IF xFalha THEN
	CASE wFalha OF
		16#0:
			sStatusConexao := 'Inversor Offline';
			xInversorOnline := FALSE;
		16#1080:
			sStatusConexao := 'Tempo Limite Backup/Restauração';
		16#1081:
			sStatusConexao := 'Falha na classificação do ID';
		16#2281:
			sStatusConexao := 'Calibração';
		16#2310:
			sStatusConexao := 'Sobrecorrente';
		16#2330:
			sStatusConexao := 'Fuga à Terra';
		16#2340:
			sStatusConexao := 'Curto-Circuito na Saída';
		16#2381:
			sStatusConexao := 'Sobrecarga no IGBT';
		16#3130:
			sStatusConexao := 'Falta de Fase na Entrada';
		16#3181:
			sStatusConexao := 'Cross Connection';
		16#3210:
			sStatusConexao := 'Sobretensão CC no Circuito intermediário';
		16#3220:
			sStatusConexao := 'Subtensão CC no Circuito intermediário';
		16#3381:
			sStatusConexao := 'Falta de Fase na Saída';
		16#4110:
			sStatusConexao := 'Temperatura alta na placa de controle';
		16#4210:
			sStatusConexao := 'Sobretemperatura estimada no IGBT';
		16#4290:
			sStatusConexao := 'Temperatura alta no módulo do inversor';
		16#42F1:
			sStatusConexao := 'Sobretemperatura no IGBT';
		16#4310:
			sStatusConexao := 'Temperatura alta no módulo de potência';
		16#4380:
			sStatusConexao := 'Diferença de temperatura IGBT';
		16#4981:
			sStatusConexao := 'Falha - Temperatura externa 1';
		16#4982:
			sStatusConexao := 'Falha - Temperatura externa 2';
		16#5090:
			sStatusConexao := 'Falha no Hardware STO';
		16#5091:
			sStatusConexao := 'STO - Safe Torque OFF';
		16#5092:
			sStatusConexao := 'Erro Lógico PU';
		16#5093:
			sStatusConexao := 'Hardware incompatível com Firmware';
		16#5094:
			sStatusConexao := 'Falha na Medição de Temperatura interna';
		16#50A0:
			sStatusConexao := 'Ventilador de Refrigeração em Falha';
		16#5681:
			sStatusConexao := 'Falha na comunicação PU';
		16#5682:
			sStatusConexao := 'Unidade de Potência Perdida';
		16#5690:
			sStatusConexao := 'Falha na Comunicação Interna';
		16#5691:
			sStatusConexao := 'Falha no Circuito de Medição';
		16#5692:
			sStatusConexao := 'Falha de Alimentação na Unidade de Potência';
		16#5693:
			sStatusConexao := 'Falha no Circuito de Medição';
		16#5696:
			sStatusConexao := 'Feedback dos Estados das Fases Incorreto';
		16#5697:
			sStatusConexao := 'Sem sinal de Feedback das Fases';
		16#6181:
			sStatusConexao := 'Versão da FPGA incompatível com o Firmware';
		16#6306:
			sStatusConexao := 'Sem sinal de Feedback das Fases';
		16#6481:
			sStatusConexao := 'Falha Interna';
		16#6487:
			sStatusConexao := 'Falha Interna';
		16#64A1:
			sStatusConexao := 'Erro de Leitura de Arquivo';
		16#64A6:
			sStatusConexao := 'Falha no programa adaptativo';
		16#64B2:
			sStatusConexao := 'Falha no conjunto de parâmetros utilizados';
		16#64E1:
			sStatusConexao := 'Erro de Sistema Operacional';
		16#6581:
			sStatusConexao := 'Falha ao salvar/carregar parâmetro';
		16#65A1:
			sStatusConexao := 'Informação requerida pelo PLC não disponpivel';
		16#6681:
			sStatusConexao := 'Perda comunicação EFB(FieldBus Integrado)';
		16#6682:
			sStatusConexao := 'Falha ao ler o arquivo EFB(FieldBus Integrado)';
		16#6683:
			sStatusConexao := 'Parâmetro EFB(FieldBus Integrado) inválido';
		16#6684:
			sStatusConexao := 'Falha ao carregar o firmware EFB(FieldBus Integrado)';
		16#6685:
			sStatusConexao := 'Falha reservada EFB(FieldBus Integrado) 1';
		16#6686:
			sStatusConexao := 'Falha reservada EFB(FieldBus Integrado) 2';
		16#6882:
			sStatusConexao := 'Falha Interna';
		16#6885:
			sStatusConexao := 'Falha Interna';
		16#7081:
			sStatusConexao := 'Perda do Painel de Controle';
		16#7082:
			sStatusConexao := 'Perda de Comunicação do Módulo I/O';
		16#7086:
			sStatusConexao := 'Sobretensão no Módulo I/O';
		16#71A2:
			sStatusConexao := 'Falha de Controle do Freio Meânico (Fechamento)';
		16#71A3:
			sStatusConexao := 'Falha de Controle do Freio Meânico (Abertura)';
		16#71A5:
			sStatusConexao := 'Freio Mecânico Travado';
		16#7121:
			sStatusConexao := 'Motor bloqueado: Carga Excessiva ou Energia Insuficiente';
		16#7181:
			sStatusConexao := 'Problema na Resistência de Frenagem';
		16#7183:
			sStatusConexao := 'Temperatura Alta na Resistência de Frenagem';
		16#7184:
			sStatusConexao := 'Curto-Circuito na Resistência de Frenagem';
		16#7191:
			sStatusConexao := 'Curto-Circuito no Chopper IGBT';
		16#7192:
			sStatusConexao := 'Temperatura Alta no Chopper IGBT';
		16#7301:
			sStatusConexao := 'Sem Feedback de Velocidade do Motor';
		16#7310:
			sStatusConexao := 'Sobrevelocidade';
		16#7381:
			sStatusConexao := 'Falha no Feedback do Encoder';
		16#73F0:
			sStatusConexao := 'Sobrefrequência';
		16#73B0:
			sStatusConexao := 'Falha na Parada de Emergência';
		16#7510:
			sStatusConexao := 'Perda de comunicação FBA A';
		16#8001:
			sStatusConexao := 'Falha de subcarga (Abaixo)';
		16#8002:
			sStatusConexao := 'Falha de subcarga (Acima)';
		16#80A0:
			sStatusConexao := 'Sinal Analógico Fora dos Limites';
		16#80B0:
			sStatusConexao := 'Falha Supervisão de Sinal 66';
		16#80B1:
			sStatusConexao := 'Falha Supervisão de Sinal 66';
		16#80B2:
			sStatusConexao := 'Falha Supervisão de Sinal 66';
		16#80B3:
			sStatusConexao := 'Falha Supervisão de Sinal 66';
		16#80B4:
			sStatusConexao := 'Falha Supervisão de Sinal 66';
		16#80B5:
			sStatusConexao := 'Falha Supervisão de Sinal 66';
		16#9081:
			sStatusConexao := 'Falha Dispotivo Externo 1';
		16#9082:
			sStatusConexao := 'Falha Dispotivo Externo 2';
		16#9083:
			sStatusConexao := 'Falha Dispotivo Externo 3';
		16#9084:
			sStatusConexao := 'Falha Dispotivo Externo 4';
		16#9085:
			sStatusConexao := 'Falha Dispotivo Externo 5';
		16#FA81:
			sStatusConexao := 'STO (Safe Torque OFF) 1 rompido';
		16#FA82:
			sStatusConexao := 'STO (Safe Torque OFF) 1 rompido';
		16#FF61:
			sStatusConexao := 'ID Run';
		16#FF81:
			sStatusConexao := 'Falha forçada FBA';
		16#FF8E:
			sStatusConexao := 'Falha forçada FBB';
		16#D100:
			sStatusConexao := 'Inversor não Consegiu Fornecer Torque Suficiente';
		16#D101:
			sStatusConexao := 'Escorregamento do Freio';
		16#D102:
			sStatusConexao := 'Velocidade abaixo do limite de segurança';
		16#D105:
			sStatusConexao := 'Velocidade do motor Excedeu o Desvio De Estado Estacionário';
		16#D108:
			sStatusConexao := 'Comando de limite de parada Frente e Ré Ativos Simultaneamente';
	END_CASE
ELSE
	IF NOT xRun AND NOT Motor.Sa.xFalha THEN
		sStatusConexao := 'Pronto para Rodar';
	ELSE
		sStatusConexao := 'Rodando';
	END_IF
	
	IF Motor.Sa.xFalha THEN
		sStatusConexao := 'Inversor OK / Falha na Partida';
	END_IF
END_IF

IF xGuardaRegistroErro THEN
	xInversorOnline := FALSE;
END_IF
END_ACTION

END_FUNCTION_BLOCK

// POUs/Comunicação/ModbusRTU/FB_ModBusRTU_ALTISTAR22
{attribute 'hide_all_locals'}
FUNCTION_BLOCK FB_ModBusRTU_ALTISTAR22
VAR_IN_OUT
	MestreModbusRTU	: ModbusRtuMasterV2_KL6x22B;
	Motor			: st_Partida;
END_VAR
VAR_INPUT
	xInicia				: BOOL;
END_VAR
VAR_OUTPUT
	//Gerais
	xTerminei				: BOOL;
	UltimoModbusErro		: ST_ModbusErrorDiagnostics;
END_VAR
VAR
	xIniciaInterno				: BOOL;	
	xTerminouLeitura			: BOOL;
	xTerminouEscrita			: BOOL;
	xSoftOnline					: BOOL;
	xGuardaRegistroErro			: BOOL;
	ControlWord					:  WORD;

	
	iRegistradorAtual			: INT := 1;
	
	wLeitura					: WORD;
	rVelocidadeAux				: WORD;
	wFalha						: WORD;
	StatusWord					: WORD;
	arLeitura					: ARRAY[1..7] OF WORD;
	arEscrita					: ARRAY[1..3] OF WORD;
	
	RegistradoresLeitura		: ARRAY[1..7] OF INT 	:= [19,20,256,257,258,259,279];		//Registradores de leitura
	RegistradoresEscrita		: ARRAY[1..3] OF INT 	:= [19,20,752];		//Registradores de escrita
	
	stateModbus					: State_Modbus;			//Variável para máquina de estados
	state						: StateWord;
	
	rt							: R_TRIG;				//Inicia vindo de fora
	ft							: F_TRIG;				//Inicio vindo de fora
	rtInicia 					: R_TRIG;				//Inicia Leitura/Escrita
	ftInicia					: F_TRIG;				//Para Leitura/Escrita
	
	tTimeout					: TIME := T#1S;			//Tempo de timeout para espera escravo 
	tonTimeout					: TON;

	xFalha					: BOOL;
	xPronto					: BOOL;
	xRodando				: BOOL;
	sStatusConexao			: STRING;
	rCorrenteL1				: REAL;
	rCorrenteL2				: REAL;
	rCorrenteL3				: REAL;
	rTempoACCAtual			: REAL;
	rTempoDECAtual			: REAL;
	
	iEndereco 			: INT;
END_VAR

IF xLicensaValida5154156 THEN
	rt(CLK := xInicia, Q =>);
	
	IF rt.Q THEN
		xIniciaInterno := TRUE;
	END_IF
	
	
	rtInicia(CLK := xIniciaInterno, Q =>);
	ftInicia(CLK := xIniciaInterno, Q =>);
	
	IF rtInicia.Q THEN
		iRegistradorAtual	:= 1;
		xTerminei			:= FALSE;
		
		//Quando inicia a leitura, não terminou de ler nenhum
		xTerminouLeitura	:= FALSE;
		xTerminouEscrita	:= FALSE;
		
		stateModbus := State_Modbus.Inicia;
	END_IF
	
	IF ftInicia.Q  THEN
		xIniciaInterno := FALSE;
		xInicia := FALSE;
		iRegistradorAtual := 1;
		xTerminei := TRUE;
		MestreModbusRTU.ReadRegs(Execute := FALSE);
		MestreModbusRTU.WriteRegs(Execute := FALSE);
	END_IF
	
	EspelhoEntradas();
	
	Leitura();
	
	Estados();
	
	ExecutaEstados();
	
	Status();
	
	EspelhoSaidas();
	
	Escrita();
	
	tonTimeOut(IN:= MestreModbusRTU.BUSY, PT:= T#10S, Q=> , ET=> );
	
	IF tonTimeOut.Q THEN
		//xIniciaInterno := FALSE;
		//xInicia := FALSE;
	END_IF

ELSE
	ValidaLicensa();
END_IF

ACTION Escrita:
CASE stateModbus OF
	
	State_Modbus.Inicia:
		IF xIniciaInterno THEN
			MestreModbusRTU.ReadRegs(Execute := FALSE);
			MestreModbusRTU.WriteSingleCoil(Execute := FALSE);

			//Se não terminou de ler corrente, fica lendo a corrente	
			IF NOT xTerminouLeitura THEN
				stateModbus := State_Modbus.Leitura;
			ELSE
				IF NOT xTerminouEscrita THEN
					stateModbus := State_Modbus.Escrita;
				END_IF
			END_IF;

			IF xTerminouLeitura AND xTerminouEscrita THEN
				xIniciaInterno := FALSE;
				xTerminei := TRUE;
			END_IF
		END_IF
			
	State_Modbus.Escrita:
	
		MestreModbusRTU.WriteSingleRegister(
			UnitID      := TO_BYTE(iEndereco),                 					// Endereço do equipamento escravo na rede Modbus
			Quantity    := 1,                									// Quantidade de WORDs a serem lidas
			MBAddr      := TO_WORD(RegistradoresEscrita[iRegistradorAtual]),	// Endereço Modbus. Onde 0 = Holding Register 40001
			cbLength    := SIZEOF(arEscrita[iRegistradorAtual]), 				// Quantidade de bytes a serem lidos
			pMemoryAddr := ADR(arEscrita[iRegistradorAtual]),					// Ponteiro para o array que receberá os dados lidos
			Execute     := TRUE,              									// Comando para executar o comando    
			Timeout     := tTimeout               								// Tempo de espera da resposta do escravo
		);

		IF NOT MestreModbusRTU.BUSY THEN
			IF MestreModbusRTU.Error THEN
				//Se deu erro cai fora
						xTerminouLeitura	:= TRUE;
						xTerminouEscrita	:= TRUE;
						
						stateModbus := State_Modbus.Inicia;
						xIniciaInterno := FALSE;
						
						xGuardaRegistroErro := TRUE;
			END_IF
			
			MestreModbusRTU.WriteSingleRegister(Execute := FALSE);
	
			stateModbus := State_Modbus.Inicia;		
			
			iRegistradorAtual := iRegistradorAtual + 1;	
			
			IF iRegistradorAtual > 3 THEN
				stateModbus := State_Modbus.Inicia;
				iRegistradorAtual := 1;
				xTerminouEscrita	:= TRUE;
				
				xGuardaRegistroErro := FALSE;
			END_IF

		END_IF 
END_CASE
END_ACTION

ACTION EspelhoEntradas:




arEscrita[1]	:= REAL_TO_WORD(Motor.Config.inversor.ACC);
arEscrita[2]	:= REAL_TO_WORD(Motor.Config.inversor.DEC);
arEscrita[3]	:= ControlWord;
iEndereco		:= Motor.En.i;

IF arEscrita[1] = 0 THEN
	arEscrita[1] := 1;
END_IF
END_ACTION

ACTION EspelhoSaidas:
StatusWord				:= arLeitura[3];
wFalha					:= arLeitura[7];

CASE wFalha OF
		1:
			Motor.Sa.sUltimoErro := 'Subcarga do Motor (Subcorrente) [UCF]';
		2:
			Motor.Sa.sUltimoErro := 'Sobrecorrente do Motor [OCF]';
		3:
			Motor.Sa.sUltimoErro := 'Desequilibrio de Fase [PHBD]';
		4:
			Motor.Sa.sUltimoErro := 'Detec. Corrente de Fuga à Terra Falha [GRDF]';
		5:
			Motor.Sa.sUltimoErro := 'Sobrecarga do Motor [OLF]';
		6:
			Motor.Sa.sUltimoErro := 'Temperatura Excessiva do Motor [OTF]';
		7:
			Motor.Sa.sUltimoErro := 'Falha Dectada de Sobreaquecimento [OHF]';
		8:
			Motor.Sa.sUltimoErro := 'Inversão de Fase [PIF]';
		9:
			Motor.Sa.sUltimoErro := 'Perda de Fase da Rede [PHF]';
		10:
			Motor.Sa.sUltimoErro := 'Subtensão ou Falta de Tensão [USF]';
		11:
			Motor.Sa.sUltimoErro := 'Sobretensão [OSF]';
		12:
			Motor.Sa.sUltimoErro := 'Falha Detectada de Tempo de Partida [STF]';
		13:
			Motor.Sa.sUltimoErro := 'Números de Partidas Excedido [SNBF]';
		14:
			Motor.Sa.sUltimoErro := 'Tiristor em Curto ou Conexão Incorreta [SSCR]';
		15:
			Motor.Sa.sUltimoErro := 'Falha Externa Detectada [ETF]';
		16:
			Motor.Sa.sUltimoErro := 'Falha Interna Detectada [INF]';
		17:
			Motor.Sa.sUltimoErro := 'Intervalo de Tempo Modbus [SLF]';
		18:
			Motor.Sa.sUltimoErro := 'Trap Code [TRAP]';
		19:
			Motor.Sa.sUltimoErro := 'Curto Circuito [SCF]';
		20:
			Motor.Sa.sUltimoErro := 'Falha Dectada Contador de By-Pass [BPF]';
		21:
			Motor.Sa.sUltimoErro := 'Config. Inválida na Energização [CFF]';
END_CASE

UltimoModbusErro			:= MestreModbusRTU.ErrorDiagnostics;
Motor.Sa.sStatusConexao		:= sStatusConexao;
Motor.En.xContatoFalhaSoft	:= xFalha AND NOT Motor.Config.xBypassRede;
Motor.Config.xTemSoft		:= TRUE;
Motor.En.xSoftOnline		:= xSoftOnline;

rTempoACCAtual			:= WORD_TO_REAL(arLeitura[1]);
rTempoDECAtual			:= WORD_TO_REAL(arLeitura[2]);
Motor.Sa.rCorrente		:= WORD_TO_REAL(arLeitura[4]);
rCorrenteL2				:= WORD_TO_REAL(arLeitura[5]);
rCorrenteL3				:= WORD_TO_REAL(arLeitura[6]);
END_ACTION

ACTION Estados:
//Rdy
IF StatusWord.0 THEN
	xPronto	:= TRUE;
ELSE
	xPronto	:= FALSE;
END_IF

//Run
IF StatusWord.1 THEN
	xRodando := TRUE;
ELSE
	xRodando := FALSE;
END_IF

//Falha
IF StatusWord.2 OR NOT StatusWord.0 THEN
	xFalha	:= TRUE;
ELSE
	xFalha	:= FALSE;
END_IF

StatusWord.0;
StatusWord.1;
StatusWord.2;
StatusWord.3;
StatusWord.4;
StatusWord.5;
StatusWord.6;
StatusWord.7;
StatusWord.8;
StatusWord.9;
StatusWord.10;
StatusWord.11;
StatusWord.12;
StatusWord.13;
StatusWord.14;
StatusWord.15;
END_ACTION

ACTION ExecutaEstados:
IF Motor.Sa.xCmdFwd THEN
	ControlWord := 1;
END_IF

IF NOT Motor.Sa.xCmdFwd THEN
	ControlWord := 0;
END_IF

IF Motor.Sa.xCmdFwd AND Motor.En.xReset THEN
	ControlWord := 9;
ELSIF NOT Motor.Sa.xCmdFwd AND Motor.En.xReset THEN
	ControlWord := 8;
END_IF

ControlWord.0;
ControlWord.1;
ControlWord.2;
ControlWord.3;
ControlWord.4;
ControlWord.5;
ControlWord.6;
ControlWord.7;
ControlWord.8;
ControlWord.9;
ControlWord.10;
ControlWord.11;
ControlWord.12;
ControlWord.13;
ControlWord.14;
ControlWord.15;
END_ACTION

ACTION Leitura:
CASE stateModbus OF
	
	State_Modbus.Inicia:
		IF xIniciaInterno THEN
			MestreModbusRTU.ReadRegs(Execute := FALSE);
			MestreModbusRTU.WriteSingleCoil(Execute := FALSE);

			//Se não terminou de ler corrente, fica lendo a corrente	
			IF NOT xTerminouLeitura THEN
				stateModbus := State_Modbus.Leitura;
			ELSE
				IF NOT xTerminouEscrita THEN
					stateModbus := State_Modbus.Escrita;
				END_IF
			END_IF;

			IF xTerminouLeitura AND xTerminouEscrita THEN
				xIniciaInterno := FALSE;
				xTerminei := TRUE;
			END_IF
		END_IF
		


	//Leitura
	State_Modbus.Leitura:
		
		MestreModbusRTU.ReadRegs(
			UnitID      := TO_BYTE(iEndereco),                 					// Endereço do equipamento escravo na rede Modbus
			Quantity    := 1,                									// Quantidade de WORDs a serem lidas
			MBAddr      := TO_WORD(RegistradoresLeitura[iRegistradorAtual]),	// Endereço Modbus. Onde 0 = Holding Register 40001
			cbLength    := SIZEOF(arLeitura[iRegistradorAtual]), 									// Quantidade de bytes a serem lidos
			pMemoryAddr := ADR(arLeitura[iRegistradorAtual]),    									// Ponteiro para o array que receberá os dados lidos
			Execute     := TRUE,              									// Comando para executar o comando    
			Timeout     := tTimeout               								// Tempo de espera da resposta do escravo
		);
	
			IF NOT MestreModbusRTU.BUSY THEN
				IF MestreModbusRTU.Error THEN
					//Se deu erro cai fora
						xTerminouLeitura	:= TRUE;
						xTerminouEscrita	:= TRUE;
						
						stateModbus := State_Modbus.Inicia;
						xIniciaInterno := FALSE;
						
						xGuardaRegistroErro := TRUE;
				END_IF

				MestreModbusRTU.ReadRegs(Execute := FALSE);
			
				iRegistradorAtual := iRegistradorAtual + 1;	
		
				stateModbus := State_Modbus.Inicia;		
				
				IF iRegistradorAtual > 7  THEN
					stateModbus := State_Modbus.Escrita;
					iRegistradorAtual := 1;
					xTerminouLeitura := TRUE;
				END_IF
			END_IF 
			
END_CASE
END_ACTION

ACTION Leitura_Escrita:
CASE stateModbus OF
	
	State_Modbus.Inicia:
		IF xIniciaInterno THEN
			MestreModbusRTU.ReadRegs(Execute := FALSE);
			MestreModbusRTU.WriteSingleCoil(Execute := FALSE);

			//Se não terminou de ler corrente, fica lendo a corrente	
			IF NOT xTerminouLeitura THEN
				stateModbus := State_Modbus.Leitura;
			ELSE
				IF NOT xTerminouEscrita THEN
					stateModbus := State_Modbus.Escrita;
				END_IF
			END_IF;

			IF xTerminouLeitura AND xTerminouEscrita THEN
				xIniciaInterno := FALSE;
				xTerminei := TRUE;
			END_IF
		END_IF
		


	//Leitura
	State_Modbus.Leitura:
		
		MestreModbusRTU.ReadRegs(
			UnitID      := TO_BYTE(iEndereco),                 					// Endereço do equipamento escravo na rede Modbus
			Quantity    := 1,                									// Quantidade de WORDs a serem lidas
			MBAddr      := TO_WORD(RegistradoresLeitura[iRegistradorAtual]),	// Endereço Modbus. Onde 0 = Holding Register 40001
			cbLength    := SIZEOF(wLeitura), 									// Quantidade de bytes a serem lidos
			pMemoryAddr := ADR(wLeitura),    									// Ponteiro para o array que receberá os dados lidos
			Execute     := TRUE,              									// Comando para executar o comando    
			Timeout     := tTimeout               								// Tempo de espera da resposta do escravo
		);
	
			IF NOT MestreModbusRTU.BUSY THEN
				IF MestreModbusRTU.Error THEN
					//Se deu erro cai fora
						xTerminouLeitura	:= TRUE;
						xTerminouEscrita	:= TRUE;
						
						stateModbus := State_Modbus.Inicia;
						xIniciaInterno := FALSE;
				END_IF

				MestreModbusRTU.ReadRegs(Execute := FALSE);
				
				arLeitura[iRegistradorAtual] := wLeitura;
			
				iRegistradorAtual := iRegistradorAtual + 1;	
		
				stateModbus := State_Modbus.Inicia;		
				
				IF iRegistradorAtual > 7  THEN
					stateModbus := State_Modbus.Escrita;
					iRegistradorAtual := 1;
					xTerminouLeitura := TRUE;
				END_IF
			END_IF 
			
	State_Modbus.Escrita:
	
		MestreModbusRTU.WriteSingleRegister(
			UnitID      := TO_BYTE(iEndereco),                 					// Endereço do equipamento escravo na rede Modbus
			Quantity    := 1,                									// Quantidade de WORDs a serem lidas
			MBAddr      := TO_WORD(RegistradoresEscrita[iRegistradorAtual]),	// Endereço Modbus. Onde 0 = Holding Register 40001
			cbLength    := SIZEOF(arEscrita[iRegistradorAtual]), 				// Quantidade de bytes a serem lidos
			pMemoryAddr := ADR(arEscrita[iRegistradorAtual]),					// Ponteiro para o array que receberá os dados lidos
			Execute     := TRUE,              									// Comando para executar o comando    
			Timeout     := tTimeout               								// Tempo de espera da resposta do escravo
		);

		IF NOT MestreModbusRTU.BUSY THEN
			IF MestreModbusRTU.Error THEN
				//Se deu erro cai fora
						xTerminouLeitura	:= TRUE;
						xTerminouEscrita	:= TRUE;
						
						stateModbus := State_Modbus.Inicia;
						xIniciaInterno := FALSE;
			END_IF
			
			MestreModbusRTU.WriteSingleRegister(Execute := FALSE);
	
			stateModbus := State_Modbus.Inicia;		
			
			iRegistradorAtual := iRegistradorAtual + 1;	
			
			IF iRegistradorAtual > 3 THEN
				stateModbus := State_Modbus.Inicia;
				iRegistradorAtual := 1;
				xTerminouEscrita	:= TRUE;
			END_IF

		END_IF 
END_CASE
END_ACTION

ACTION Status:
IF xFalha THEN
	CASE wFalha OF
		1:
			sStatusConexao := 'Subcarga do Motor (Subcorrente) [UCF]';
		2:
			sStatusConexao := 'Sobrecorrente do Motor [OCF]';
		3:
			sStatusConexao := 'Desequilibrio de Fase [PHBD]';
		4:
			sStatusConexao := 'Detec. Corrente de Fuga à Terra Falha [GRDF]';
		5:
			sStatusConexao := 'Sobrecarga do Motor [OLF]';
		6:
			sStatusConexao := 'Temperatura Excessiva do Motor [OTF]';
		7:
			sStatusConexao := 'Falha Dectada de Sobreaquecimento [OHF]';
		8:
			sStatusConexao := 'Inversão de Fase [PIF]';
		9:
			sStatusConexao := 'Perda de Fase da Rede [PHF]';
		10:
			sStatusConexao := 'Subtensão ou Falta de Tensão [USF]';
		11:
			sStatusConexao := 'Sobretensão [OSF]';
		12:
			sStatusConexao := 'Falha Detectada de Tempo de Partida [STF]';
		13:
			sStatusConexao := 'Números de Partidas Excedido [SNBF]';
		14:
			sStatusConexao := 'Tiristor em Curto ou Conexão Incorreta [SSCR]';
		15:
			sStatusConexao := 'Falha Externa Detectada [ETF]';
		16:
			sStatusConexao := 'Falha Interna Detectada [INF]';
		17:
			sStatusConexao := 'Intervalo de Tempo Modbus [SLF]';
		18:
			sStatusConexao := 'Trap Code [TRAP]';
		19:
			sStatusConexao := 'Curto Circuito [SCF]';
		20:
			sStatusConexao := 'Falha Dectada Contador de By-Pass [BPF]';
		21:
			sStatusConexao := 'Config. Inválida na Energização [CFF]';
	END_CASE
ELSE
	IF xPronto AND NOT xRodando THEN
		sStatusConexao := 'Pronto';
	ELSIF xPronto AND xRodando THEN
		sStatusConexao := 'Rodando';
	END_IF
END_IF

xSoftOnline := NOT xGuardaRegistroErro;
END_ACTION

END_FUNCTION_BLOCK

// POUs/Comunicação/ModbusRTU/FB_ModBusRTU_ATV320
//{attribute 'hide_all_locals'}
FUNCTION_BLOCK FB_ModBusRTU_ATV320
VAR_IN_OUT
	MestreModbusRTU	: ModbusRtuMasterV2_KL6x22B;
	Motor			: st_Partida;
END_VAR
VAR_INPUT
	xInicia				: BOOL;
END_VAR
VAR_OUTPUT
	//Gerais
	xTerminei				: BOOL;
	UltimoModbusErro		: ST_ModbusErrorDiagnostics;
END_VAR
VAR
	xIniciaInterno				: BOOL;	
	xTerminouLeitura			: BOOL;
	xTerminouEscrita			: BOOL;
	xFalha						: BOOL;
	xInversorOnline				: BOOL;
	ControlWord					: ARRAY[0..15] OF BOOL;

	
	iRegistradorAtual			: INT := 1;
	iEndereco 					: INT;
	
	wDriveState					: WORD;
	wLeitura					: WORD;
	rVelocidadeAux				: WORD;
	wFalha						: WORD;
	StatusWord					: WORD;
	arLeitura					: ARRAY[1..13] OF WORD;
	arEscrita					: ARRAY[1..3] OF WORD;
	
	RegistradoresLeitura		: ARRAY[1..13] OF INT 	:= [3204,3205,3208,3209,3211,3240,7210,7121,3202,8604,9001,9002,9630];		//Registradores de leitura
	RegistradoresEscrita		: ARRAY[1..3] OF INT 	:= [8602,9001,9002];		//Registradores de escrita
	
	stateModbus					: State_Modbus;			//Variável para máquina de estados
	state						: StateWord;
	
	rt							: R_TRIG;				//Inicia vindo de fora
	ft							: F_TRIG;				//Inicio vindo de fora
	rtInicia 					: R_TRIG;				//Inicia Leitura/Escrita
	ftInicia					: F_TRIG;				//Para Leitura/Escrita
	
	tTimeout					: TIME := T#1S;			//Tempo de timeout para espera escravo 
	tonTimeOut					: Tc2_Standard.TON;
	
	sStatusConexao				: STRING;
	sUltimoErro					: STRING;
	
	rRampaACCAtual			: REAL;
	rRampaDCCAtual			: REAL;
	
	rPotencia				: REAL;

END_VAR

IF xLicensaValida5154156 THEN
	
	rt(CLK := xInicia, Q =>);
	
	IF rt.Q THEN
		xIniciaInterno := TRUE;
	END_IF
	
	
	rtInicia(CLK := xIniciaInterno, Q =>);
	ftInicia(CLK := xIniciaInterno, Q =>);
	
	IF rtInicia.Q THEN
		iRegistradorAtual	:= 1;
		xTerminei			:= FALSE;
		
		//Quando inicia a leitura, não terminou de ler nenhum
		xTerminouLeitura	:= FALSE;
		xTerminouEscrita	:= FALSE;
		
		stateModbus := State_Modbus.Inicia;
	END_IF
	
	IF ftInicia.Q  THEN
		xIniciaInterno := FALSE;
		xInicia			:= FALSE;
		iRegistradorAtual := 1;
		xTerminei := TRUE;
		MestreModbusRTU.ReadRegs(Execute := FALSE);
		MestreModbusRTU.WriteRegs(Execute := FALSE);
	END_IF
	
	
	EspelhoEntradas();
	
	Leitura();
	
	Estados();
	
	//ExecutaEstados();
	
	Status();
	
	EspelhoSaidas();
	
	Escrita();
	
	tonTimeOut(IN:= MestreModbusRTU.BUSY, PT:= T#10S, Q=> , ET=> );
	
	IF tonTimeOut.Q THEN
		xIniciaInterno := FALSE;
		xInversorOnline := FALSE;
		xInicia := FALSE;
	END_IF
	
ELSE
	ValidaLicensa();
END_IF

ACTION Escrita:
CASE stateModbus OF
	
	State_Modbus.Inicia:
		IF xIniciaInterno THEN
			MestreModbusRTU.ReadRegs(Execute := FALSE);
			MestreModbusRTU.WriteSingleCoil(Execute := FALSE);

			//Se não terminou de ler corrente, fica lendo a corrente	
			IF NOT xTerminouLeitura THEN
				stateModbus := State_Modbus.Leitura;
			ELSE
				IF NOT xTerminouEscrita THEN
					stateModbus := State_Modbus.Escrita;
				END_IF
			END_IF;

			IF xTerminouLeitura AND xTerminouEscrita THEN
				xIniciaInterno := FALSE;
				xTerminei := TRUE;
			END_IF
		END_IF
			
	State_Modbus.Escrita:
	
		MestreModbusRTU.WriteSingleRegister(
			UnitID      := TO_BYTE(iEndereco),                 					// Endereço do equipamento escravo na rede Modbus
			Quantity    := 1,                									// Quantidade de WORDs a serem lidas
			MBAddr      := TO_WORD(RegistradoresEscrita[iRegistradorAtual]),	// Endereço Modbus. Onde 0 = Holding Register 40001
			cbLength    := SIZEOF(arEscrita[iRegistradorAtual]), 				// Quantidade de bytes a serem lidos
			pMemoryAddr := ADR(arEscrita[iRegistradorAtual]),					// Ponteiro para o array que receberá os dados lidos
			Execute     := TRUE,              									// Comando para executar o comando    
			Timeout     := tTimeout               								// Tempo de espera da resposta do escravo
		);

		IF NOT MestreModbusRTU.BUSY THEN
			IF MestreModbusRTU.Error THEN
				//Se deu erro cai fora
						xTerminouLeitura	:= TRUE;
						xTerminouEscrita	:= TRUE;
						
						stateModbus := State_Modbus.Inicia;
						xIniciaInterno := FALSE;
			END_IF
			
			MestreModbusRTU.WriteSingleRegister(Execute := FALSE);
	
			stateModbus := State_Modbus.Inicia;		
			
			iRegistradorAtual := iRegistradorAtual + 1;	
			
			IF iRegistradorAtual > 3 THEN
				stateModbus := State_Modbus.Inicia;
				iRegistradorAtual := 1;
				xTerminouEscrita	:= TRUE;
			END_IF
		END_IF 
END_CASE
END_ACTION

ACTION EspelhoEntradas:


arEscrita[1]	:= INT_TO_WORD(Motor.Sa.iVelocidade);
arEscrita[2]	:= REAL_TO_WORD(Motor.Config.inversor.ACC)*10;
arEscrita[3]	:= REAL_TO_WORD(Motor.Config.inversor.DEC)*10;
iEndereco		:= Motor.En.i;
END_ACTION

ACTION EspelhoSaidas:
Motor.Sa.rCorrente			:= WORD_TO_REAL(arLeitura[1])/10;
Motor.Sa.rTorque			:= WORD_TO_REAL(arLeitura[2]);
Motor.Sa.rVoltagemEntrada	:= WORD_TO_REAL(arLeitura[3]);
Motor.Sa.rTemperaturaInver	:= WORD_TO_REAL(arLeitura[4]);
rPotencia					:= WORD_TO_REAL(arLeitura[5]);
Motor.Sa.rVelocidadeHz		:= WORD_TO_REAL(arLeitura[9])/10;
Motor.Sa.rVelocidadeRPM		:= WORD_TO_REAL(arLeitura[10]);
rRampaACCAtual				:= WORD_TO_REAL(arLeitura[11])/10;
rRampaDCCAtual				:= WORD_TO_REAL(arLeitura[12])/10;
Motor.Sa.rTemperaturaMotor	:= WORD_TO_REAL(arLeitura[13]);
Motor.En.xFalhaInversor		:= xFalha;
Motor.Sa.sStatusConexao		:= sStatusConexao;
Motor.En.xTemInversor 		:= TRUE;
Motor.En.xInversorOnline 	:= xInversorOnline;
Motor.Sa.sUltimoErro		:= sUltimoErro;


UltimoModbusErro	:= MestreModbusRTU.ErrorDiagnostics;
END_ACTION

ACTION Estados:

END_ACTION

ACTION ExecutaEstados:

END_ACTION

ACTION Leitura:
CASE stateModbus OF
	
	State_Modbus.Inicia:
		IF xIniciaInterno THEN
			MestreModbusRTU.ReadRegs(Execute := FALSE);
			MestreModbusRTU.WriteSingleCoil(Execute := FALSE);

			//Se não terminou de ler corrente, fica lendo a corrente	
			IF NOT xTerminouLeitura THEN
				stateModbus := State_Modbus.Leitura;
			ELSE
				IF NOT xTerminouEscrita THEN
					stateModbus := State_Modbus.Escrita;
				END_IF
			END_IF;

			IF xTerminouLeitura AND xTerminouEscrita THEN
				xIniciaInterno := FALSE;
				xTerminei := TRUE;
			END_IF
		END_IF
		


	//Leitura
	State_Modbus.Leitura:
		
		MestreModbusRTU.ReadRegs(
			UnitID      := TO_BYTE(iEndereco),                 					// Endereço do equipamento escravo na rede Modbus
			Quantity    := 1,                									// Quantidade de WORDs a serem lidas
			MBAddr      := TO_WORD(RegistradoresLeitura[iRegistradorAtual]),	// Endereço Modbus. Onde 0 = Holding Register 40001
			cbLength    := SIZEOF(arLeitura[iRegistradorAtual]), 									// Quantidade de bytes a serem lidos
			pMemoryAddr := ADR(arLeitura[iRegistradorAtual]),    									// Ponteiro para o array que receberá os dados lidos
			Execute     := TRUE,              									// Comando para executar o comando    
			Timeout     := tTimeout               								// Tempo de espera da resposta do escravo
		);
	
			IF NOT MestreModbusRTU.BUSY THEN
				IF MestreModbusRTU.Error THEN
					//Se deu erro cai fora
						xTerminouLeitura	:= TRUE;
						xTerminouEscrita	:= TRUE;
						
						stateModbus := State_Modbus.Inicia;
						xIniciaInterno := FALSE;
						
						arLeitura[6] := 33;
						arLeitura[8] := 0;
				END_IF

				MestreModbusRTU.ReadRegs(Execute := FALSE);
				
				//arLeitura[iRegistradorAtual] := wLeitura;
			
				iRegistradorAtual := iRegistradorAtual + 1;	
		
				stateModbus := State_Modbus.Inicia;		
				
				IF iRegistradorAtual > 13 THEN
					stateModbus := State_Modbus.Escrita;
					iRegistradorAtual := 1;
					xTerminouLeitura := TRUE;
				END_IF
			END_IF 
			
END_CASE

wDriveState					:= arLeitura[6];
StatusWord					:= arLeitura[7];
wFalha						:= arLeitura[8];
END_ACTION

ACTION Leitura_Escrita:
CASE stateModbus OF
	
	State_Modbus.Inicia:
		IF xIniciaInterno THEN
			MestreModbusRTU.ReadRegs(Execute := FALSE);
			MestreModbusRTU.WriteSingleCoil(Execute := FALSE);

			//Se não terminou de ler corrente, fica lendo a corrente	
			IF NOT xTerminouLeitura THEN
				stateModbus := State_Modbus.Leitura;
			ELSE
				IF NOT xTerminouEscrita THEN
					stateModbus := State_Modbus.Escrita;
				END_IF
			END_IF;

			IF xTerminouLeitura AND xTerminouEscrita THEN
				xIniciaInterno := FALSE;
				xTerminei := TRUE;
			END_IF
		END_IF
		


	//Leitura
	State_Modbus.Leitura:
		
		MestreModbusRTU.ReadRegs(
			UnitID      := TO_BYTE(iEndereco),                 					// Endereço do equipamento escravo na rede Modbus
			Quantity    := 1,                									// Quantidade de WORDs a serem lidas
			MBAddr      := TO_WORD(RegistradoresLeitura[iRegistradorAtual]),	// Endereço Modbus. Onde 0 = Holding Register 40001
			cbLength    := SIZEOF(wLeitura), 									// Quantidade de bytes a serem lidos
			pMemoryAddr := ADR(wLeitura),    									// Ponteiro para o array que receberá os dados lidos
			Execute     := TRUE,              									// Comando para executar o comando    
			Timeout     := tTimeout               								// Tempo de espera da resposta do escravo
		);
	
			IF NOT MestreModbusRTU.BUSY THEN
				IF MestreModbusRTU.Error THEN
					//Se deu erro cai fora
						xTerminouLeitura	:= TRUE;
						xTerminouEscrita	:= TRUE;
						
						stateModbus := State_Modbus.Inicia;
						xIniciaInterno := FALSE;
				END_IF

				MestreModbusRTU.ReadRegs(Execute := FALSE);
				
				arLeitura[iRegistradorAtual] := wLeitura;
			
				iRegistradorAtual := iRegistradorAtual + 1;	
		
				stateModbus := State_Modbus.Inicia;		
				
				IF iRegistradorAtual > 13 THEN
					stateModbus := State_Modbus.Escrita;
					iRegistradorAtual := 1;
					xTerminouLeitura := TRUE;
				END_IF
			END_IF 
			
	State_Modbus.Escrita:
	
		MestreModbusRTU.WriteSingleRegister(
			UnitID      := TO_BYTE(iEndereco),                 					// Endereço do equipamento escravo na rede Modbus
			Quantity    := 1,                									// Quantidade de WORDs a serem lidas
			MBAddr      := TO_WORD(RegistradoresEscrita[iRegistradorAtual]),	// Endereço Modbus. Onde 0 = Holding Register 40001
			cbLength    := SIZEOF(arEscrita[iRegistradorAtual]), 				// Quantidade de bytes a serem lidos
			pMemoryAddr := ADR(arEscrita[iRegistradorAtual]),					// Ponteiro para o array que receberá os dados lidos
			Execute     := TRUE,              									// Comando para executar o comando    
			Timeout     := tTimeout               								// Tempo de espera da resposta do escravo
		);

		IF NOT MestreModbusRTU.BUSY THEN
			IF MestreModbusRTU.Error THEN
				//Se deu erro cai fora
						xTerminouLeitura	:= TRUE;
						xTerminouEscrita	:= TRUE;
						
						stateModbus := State_Modbus.Inicia;
						xIniciaInterno := FALSE;
			END_IF
			
			MestreModbusRTU.WriteSingleRegister(Execute := FALSE);
	
			stateModbus := State_Modbus.Inicia;		
			
			iRegistradorAtual := iRegistradorAtual + 1;	
			
			IF iRegistradorAtual > 4 THEN
				stateModbus := State_Modbus.Inicia;
				iRegistradorAtual := 1;
				xTerminouEscrita	:= TRUE;
			END_IF

		END_IF 
END_CASE
END_ACTION

ACTION Status:
xFalha := FALSE;
xInversorOnline := TRUE;

CASE wDriveState OF
		0:
			sStatusConexao := '[Auto-tuning] (TUN)';
			xInversorOnline := FALSE;
		1:
			sStatusConexao := '[In DC inject.] (DCB)';
		2:
			sStatusConexao := '[Ready] (RDY)';
		3:
			sStatusConexao := '[Freewheel] (NST)';
		4:
			sStatusConexao := '[Drv running] (RUN)';
		5:
			sStatusConexao := '[In accel.] (ACC)';
		6:
			sStatusConexao := '[In decel.] (DEC)';
		7:
			sStatusConexao := '[Current lim.] (CLI)';
		8:
			sStatusConexao := '[Fast stop] (FST)';
		9:
			sStatusConexao := '[Mot. fluxing] (FLU)';
		10:
			sStatusConexao := '';
		11:
			sStatusConexao := '[no mains V.] (NLP)';
		12:
			sStatusConexao := '[Active PWR] (PRA)';
		13:
			sStatusConexao := '[control.stop] (CTL)';
		14:
			sStatusConexao := '[Dec. adapt.] (OBR)';
		15:
			sStatusConexao := '[Output cut] (SOC)';
		16:
			sStatusConexao := '';
		17:
			sStatusConexao := '[UnderV. al.] (USA)';
		18:
			sStatusConexao := '[In mfg. test] (TC)';
		19:
			sStatusConexao := '[in autotest] (ST)';
		20:
			sStatusConexao := '[autotest err] (FA)';
		21:
			sStatusConexao := '[Autotest OK] (OK)';
		22:
			sStatusConexao := '[eeprom test] (EP)';
		23:
			//sStatusConexao := '[In fault] (FLT)';
			
			xFalha := TRUE;
				CASE wFalha OF
					0:
						sStatusConexao := '[No fault] (NOF)';
					2:
						sStatusConexao := '[Control Eeprom] (EEF1)';
					3:
						sStatusConexao := '[Incorrect config.] (CFF)';
					4:
						sStatusConexao := '[Invalid config.] (CFI)';
					5:
						sStatusConexao := '[Modbus com.] (SLF1)';
					6:
						sStatusConexao := '[int. com.link] (ILF)';
					7:
						sStatusConexao := '[Com. network] (CNF)';
					8:
						sStatusConexao := '[External flt-LI/Bit] (EPF1)';
					9:
						sStatusConexao := '[Overcurrent] (OCF)';
					10:
						sStatusConexao := '[Precharge] (CRF1)';
					11:
						sStatusConexao := '[Speed fdback loss] (SPF)';
					12:
						sStatusConexao := '[Load slipping] (ANF)';
					16:
						sStatusConexao := '[Drive overheat] (OHF)';
					17:
						sStatusConexao := '[Motor overload] (OLF)';
					18:
						sStatusConexao := '[Overbraking] (OBF)';
					19:
						sStatusConexao := '[Mains overvoltage] (OSF)';
					20:
						sStatusConexao := '[1 output phase loss] (OPF1)';
					21:
						sStatusConexao := '[Input phase loss] (PHF)';
					22:
						sStatusConexao := '[Undervoltage] (USF)';
					23:
						sStatusConexao := '[Motor short circuit] (SCF1)';
					24:
						sStatusConexao := '[Overspeed] (SOF)';
					25:
						sStatusConexao := '[Auto-tuning ] (TNF)';
					26:
						sStatusConexao := '[Rating error] (INF1)';
					27:
						sStatusConexao := '[PWR Calib.] (INF2)';
					28:
						sStatusConexao := '[Int.serial link] (INF3)';
					29:
						sStatusConexao := '[Int.Mfg area] (INF4)';
					30:
						sStatusConexao := '[Power Eeprom] (EEF2)';
					32:
						sStatusConexao := '[Ground short circuit] (SCF3)';
					33:
						sStatusConexao := '[3out ph loss] (OPF2)';
					34:
						sStatusConexao := '[CAN com.] (COF)';
					35:
						sStatusConexao := '[Brake control] (BLF)';
					38:
						sStatusConexao := '[External fault com.] (EPF2)';
					41:
						sStatusConexao := '[Brake feedback] (BRF)';
					42:
						sStatusConexao := '[PC com.] (SLF2)';
					44:
						sStatusConexao := '[Torque/current lim] (SSF)';
					45:
						sStatusConexao := '[HMI com.] (SLF3)';
					49:
						sStatusConexao := '[LI6=PTC probe] (PTFL)';
					50:
						sStatusConexao := '[PTC fault] (OTFL)';
					51:
						sStatusConexao := '[Internal- I measure] (INF9)';
					52:
						sStatusConexao := '[Internal-mains circuit] (INFA)';
					53:
						sStatusConexao := '[Internal- th. sensor] (INFB)';
					54:
						sStatusConexao := '[IGBT overheat] (TJF)';
					55:
						sStatusConexao := '[IGBT short circuit] (SCF4)';
					56:
						sStatusConexao := '[Motor short circuit] (SCF5)';
					58:
						sStatusConexao := '[Out. contact. stuck] (FCF1)';
					59:
						sStatusConexao := '[Out. contact. open.] (FCF2)';
					64:
						sStatusConexao := '[input contactor] (LCF)';
					67:
						sStatusConexao := '[IGBT desaturation] (HDF)';
					68:
						sStatusConexao := '[Internal-option] (INF6)';
					69:
						sStatusConexao := '[internal- CPU ] (INFE)';
					71:
						sStatusConexao := '[AI3 4-20mA loss] (LFF3)';
					73:
						sStatusConexao := '[Cards pairing] (HCF)';
					76:
						sStatusConexao := '[Load fault] (DLF)';
					77:
						sStatusConexao := '[Bad conf] (CFI2)';
					99:
						sStatusConexao := '[Ch.sw. fault] (CSF)';
					100:
						sStatusConexao := '[Pr.Underload.Flt] (ULF)';
					101:
						sStatusConexao := '[Proc.Overload Flt] (OLC)';
					105:
						sStatusConexao := '[Angle error] (ASF)';
					107:
						sStatusConexao := '[Safety fault] (SAFF)';
					108:
						sStatusConexao := '[FB fault] (FBE)';
					109:
						sStatusConexao := '[FB stop flt.] (FBES)';	
				END_CASE
		24:
			sStatusConexao := '';
		25:
			sStatusConexao := '[DCP] (DCP)';
		26:
			sStatusConexao := '';
		27:
			sStatusConexao := '';
		28:
			sStatusConexao := '[SS1 active] (SS1)';
		29:
			sStatusConexao := '[SLS active] (SLS)';
		30:
			sStatusConexao := '[STO active] (STO)';
		31:
			sStatusConexao := '[None] (SMS)';
		32:
			sStatusConexao := '[None] (GDL)';
		33:
			sStatusConexao := 'Inversor Offline';
			xInversorOnline := FALSE;
	END_CASE


CASE wFalha OF
		0:
			sUltimoErro := '[No fault] (NOF)';
		2:
			sUltimoErro := '[Control Eeprom] (EEF1)';
		3:
			sUltimoErro := '[Incorrect config.] (CFF)';
		4:
			sUltimoErro := '[Invalid config.] (CFI)';
		5:
			sUltimoErro := '[Modbus com.] (SLF1)';
		6:
			sUltimoErro := '[int. com.link] (ILF)';
		7:
			sUltimoErro := '[Com. network] (CNF)';
		8:
			sUltimoErro := '[External flt-LI/Bit] (EPF1)';
		9:
			sUltimoErro := '[Overcurrent] (OCF)';
		10:
			sUltimoErro := '[Precharge] (CRF1)';
		11:
			sUltimoErro := '[Speed fdback loss] (SPF)';
		12:
			sUltimoErro := '[Load slipping] (ANF)';
		16:
			sUltimoErro := '[Drive overheat] (OHF)';
		17:
			sUltimoErro := '[Motor overload] (OLF)';
		18:
			sUltimoErro := '[Overbraking] (OBF)';
		19:
			sUltimoErro := '[Mains overvoltage] (OSF)';
		20:
			sUltimoErro := '[1 output phase loss] (OPF1)';
		21:
			sUltimoErro := '[Input phase loss] (PHF)';
		22:
			sUltimoErro := '[Undervoltage] (USF)';
		23:
			sUltimoErro := '[Motor short circuit] (SCF1)';
		24:
			sUltimoErro := '[Overspeed] (SOF)';
		25:
			sUltimoErro := '[Auto-tuning ] (TNF)';
		26:
			sUltimoErro := '[Rating error] (INF1)';
		27:
			sUltimoErro := '[PWR Calib.] (INF2)';
		28:
			sUltimoErro := '[Int.serial link] (INF3)';
		29:
			sUltimoErro := '[Int.Mfg area] (INF4)';
		30:
			sUltimoErro := '[Power Eeprom] (EEF2)';
		32:
			sUltimoErro := '[Ground short circuit] (SCF3)';
		33:
			sUltimoErro := '[3out ph loss] (OPF2)';
		34:
			sUltimoErro := '[CAN com.] (COF)';
		35:
			sUltimoErro := '[Brake control] (BLF)';
		38:
			sUltimoErro := '[External fault com.] (EPF2)';
		41:
			sUltimoErro := '[Brake feedback] (BRF)';
		42:
			sUltimoErro := '[PC com.] (SLF2)';
		44:
			sUltimoErro := '[Torque/current lim] (SSF)';
		45:
			sUltimoErro := '[HMI com.] (SLF3)';
		49:
			sUltimoErro := '[LI6=PTC probe] (PTFL)';
		50:
			sUltimoErro := '[PTC fault] (OTFL)';
		51:
			sUltimoErro := '[Internal- I measure] (INF9)';
		52:
			sUltimoErro := '[Internal-mains circuit] (INFA)';
		53:
			sUltimoErro := '[Internal- th. sensor] (INFB)';
		54:
			sUltimoErro := '[IGBT overheat] (TJF)';
		55:
			sUltimoErro := '[IGBT short circuit] (SCF4)';
		56:
			sUltimoErro := '[Motor short circuit] (SCF5)';
		58:
			sUltimoErro := '[Out. contact. stuck] (FCF1)';
		59:
			sUltimoErro := '[Out. contact. open.] (FCF2)';
		64:
			sUltimoErro := '[input contactor] (LCF)';
		67:
			sUltimoErro := '[IGBT desaturation] (HDF)';
		68:
			sUltimoErro := '[Internal-option] (INF6)';
		69:
			sUltimoErro := '[internal- CPU ] (INFE)';
		71:
			sUltimoErro := '[AI3 4-20mA loss] (LFF3)';
		73:
			sUltimoErro := '[Cards pairing] (HCF)';
		76:
			sUltimoErro := '[Load fault] (DLF)';
		77:
			sUltimoErro := '[Bad conf] (CFI2)';
		99:
			sUltimoErro := '[Ch.sw. fault] (CSF)';
		100:
			sUltimoErro := '[Pr.Underload.Flt] (ULF)';
		101:
			sUltimoErro := '[Proc.Overload Flt] (OLC)';
		105:
			sUltimoErro := '[Angle error] (ASF)';
		107:
			sUltimoErro := '[Safety fault] (SAFF)';
		108:
			sUltimoErro := '[FB fault] (FBE)';
		109:
			sUltimoErro := '[FB stop flt.] (FBES)';
	
	END_CASE
END_ACTION

END_FUNCTION_BLOCK

// POUs/Partida/Test/FB_Partida_Teste
FUNCTION_BLOCK FB_Partida_Teste EXTENDS TcUnit.FB_TestSuite
VAR
	stMotor					: st_Partida;
	stMotorVazio			: st_Partida;
	Partida					: FB_Partida;
	i						: INT;
	xTerminouTodos			: BOOL;
	xFaltaSoOsQueTemTempo	: BOOL;
	xComecou				: BOOL;

	tonFalha		: ton;
	tonBypass		: ton;
	tonProxPartida	: ton;
	tonReversao		: TON;

	EstadoReversao : INT := 0;

	xAux : BOOL;

END_VAR

Velocidade();
Interlocks();
Falhas();
Bypasses();
ProxPartida();
Emergencia();
Reversao();

METHOD PRIVATE Bypasses
VAR
END_VAR
IF TEST_ORDERED('bypasses') THEN

	IF NOT xFaltaSoOsQueTemTempo THEN

		stMotor := stMotorVazio;

		//config inicial da partida
		Partida(stMotor := stMotor);

		stMotor.En.xEmergenciaOK		:= TRUE;
		stMotor.En.xDisjuntorOK			:= TRUE;
		stMotor.En.xContatorLigado		:= TRUE;
		stMotor.En.xAutomaticoManual	:= TRUE;
		stMotor.En.xBloqueado			:= FALSE;

		Partida(stMotor := stMotor);
		//final ocnfig inicial da partida

		stMotor.Config.xByPassDisjuntor	:= TRUE;
		stMotor.En.xDisjuntorOK			:= FALSE;
		Partida(stMotor := stMotor);

		AssertEquals_BOOL
			(
				Expected := FALSE,
					Actual := stMotor.Sa.xFalha,
					Message := ('xFalha foi acionado mesmo o bypass do disjuntor estando acionado'));

		stMotor.Config.xByPassDisjuntor	:= FALSE;
		stMotor.En.xDisjuntorOK			:= TRUE;
		Partida(stMotor := stMotor);

		//freio
		stMotor.Config.xTemFreio	:= TRUE;
		stMotor.Config.xBypassFreio	:= TRUE;
		stMotor.En.xFreioOK			:= FALSE;
		Partida(stMotor := stMotor);

		AssertEquals_BOOL
			(
				Expected := FALSE,
					Actual := stMotor.Sa.xFalha,
					Message := ('xFalha foi acionado mesmo o bypass do freio estando acionado'));

		stMotor.Config.xTemFreio	:= FALSE;
		stMotor.Config.xBypassFreio	:= FALSE;
		stMotor.En.xFreioOK			:= FALSE;
		Partida(stMotor := stMotor);

		//inversor em falha
		stMotor.En.xTemInversor		:= TRUE;
		stMotor.Config.xBypassRede	:= TRUE;
		stMotor.En.xFalhaInversor	:= TRUE;
		Partida(stMotor := stMotor);

		AssertEquals_BOOL
			(
				Expected := FALSE,
					Actual := stMotor.Sa.xFalha,
					Message := ('xFalha foi acionado mesmo o bypass da rede estando acionado quando o inversor esta em falha'));

		stMotor.En.xTemInversor		:= FALSE;
		stMotor.Config.xBypassRede	:= FALSE;
		stMotor.En.xFalhaInversor	:= FALSE;
		Partida(stMotor := stMotor);

		//inversor em offline
		stMotor.En.xTemInversor		:= TRUE;
		stMotor.Config.xBypassRede	:= TRUE;
		stMotor.En.xInversorOnline	:= FALSE;
		Partida(stMotor := stMotor);

		AssertEquals_BOOL
			(
				Expected := FALSE,
					Actual := stMotor.Sa.xFalha,
					Message := ('xFalha foi acionado mesmo o bypass da rede estando acionado quando o inversor esta em offline'));

		stMotor.En.xTemInversor		:= FALSE;
		stMotor.Config.xBypassRede	:= FALSE;
		stMotor.En.xInversorOnline	:= FALSE;
		Partida(stMotor := stMotor);

		xFaltaSoOsQueTemTempo := TRUE;
	END_IF

	stMotor.En.xLigaAuto					:= TRUE;
	stMotor.En.xContatorLigado				:= FALSE;
	stMotor.Config.rTempoFeedBackContator	:= 1.5;
	stMotor.Config.xByPassContator			:= TRUE;
	stMotor.En.xEmergenciaOK				:= TRUE;
	stMotor.En.xDisjuntorOK					:= TRUE;
	stMotor.En.xAutomaticoManual			:= TRUE;
	Partida(stMotor := stMotor);

	tonBypass(IN := stMotor.Sa.xCmdFwd, PT := REAL_TO_TIME(stMotor.Config.rTempoFeedBackContator * 1000), Q =>, ET =>);

	IF tonBypass.q THEN
		Partida(stMotor := stMotor);

		AssertEquals_BOOL
			(
				Expected := FALSE,
					Actual := stMotor.Sa.xFalha,
					Message := ('xFalha foi acionado quando o bypass do contato estava acionado'));

		xTerminouTodos := TRUE;
	END_IF

	IF xTerminouTodos THEN
		xTerminouTodos			:= FALSE;
		xFaltaSoOsQueTemTempo	:= FALSE;

		TEST_FINISHED();
	END_IF

END_IF
END_METHOD

METHOD PRIVATE Emergencia
VAR
END_VAR
IF TEST_ORDERED('Emergencia') THEN

	stMotor := stMotorVazio;

	//config inicial da partida
	Partida(stMotor := stMotor);

	stMotor.En.xEmergenciaOK		:= FALSE;
	stMotor.En.xLigaAuto			:= TRUE;
	stMotor.En.xContatorLigado		:= TRUE;
	stMotor.En.xDisjuntorOK			:= TRUE;
	stMotor.En.xAutomaticoManual	:= TRUE;
	stMotor.En.xBloqueado			:= FALSE;

	Partida(stMotor := stMotor);
	//final ocnfig inicial da partida

	AssertEquals_BOOL
		(
			Expected := FALSE,
				Actual := stMotor.Sa.xLigado,
				Message := 'xLigado acionado em emergencia');

	AssertEquals_BOOL
		(
			Expected := FALSE,
				Actual := stMotor.Sa.xCmdFwd,
				Message := 'xCmdFwd acionado em emergencia');

	AssertEquals_BOOL
		(
			Expected := FALSE,
				Actual := stMotor.Sa.xCmdRev,
				Message := 'xCmdRev acionado em emergencia');

	TEST_FINISHED();

END_IF
END_METHOD

METHOD PRIVATE Falhas
VAR
END_VAR
IF TEST_ORDERED('Falhas') THEN

	IF NOT xFaltaSoOsQueTemTempo THEN

		stMotor := stMotorVazio;

		//config inicial da partida
		Partida(stMotor := stMotor);

		stMotor.En.xEmergenciaOK		:= TRUE;
		stMotor.En.xDisjuntorOK			:= TRUE;
		stMotor.En.xContatorLigado		:= TRUE;
		stMotor.En.xAutomaticoManual	:= TRUE;
		stMotor.En.xBloqueado			:= FALSE;

		Partida(stMotor := stMotor);
		//final ocnfig inicial da partida

		stMotor.Config.xByPassDisjuntor	:= FALSE;
		stMotor.En.xDisjuntorOK			:= FALSE;
		Partida(stMotor := stMotor);

		AssertEquals_BOOL
			(
				Expected := TRUE,
					Actual := stMotor.Sa.xFalha,
					Message := ('xFalha nao foi acionado quando o disjuntor estava estava em falha'));

		stMotor.Config.xByPassDisjuntor	:= FALSE;
		stMotor.En.xDisjuntorOK			:= TRUE;
		Partida(stMotor := stMotor);

		//freio
		stMotor.Config.xTemFreio	:= TRUE;
		stMotor.En.xFreioOK			:= FALSE;
		Partida(stMotor := stMotor);

		AssertEquals_BOOL
			(
				Expected := TRUE,
					Actual := stMotor.Sa.xFalha,
					Message := ('xFalha nao foi acionado quando o xfreio estava em falha'));

		stMotor.Config.xTemFreio	:= FALSE;
		stMotor.En.xFreioOK			:= FALSE;
		Partida(stMotor := stMotor);

		//inversor em falha
		stMotor.En.xTemInversor		:= TRUE;
		stMotor.En.xFalhaInversor	:= FALSE;
		Partida(stMotor := stMotor);

		AssertEquals_BOOL
			(
				Expected := TRUE,
					Actual := stMotor.Sa.xFalha,
					Message := ('xFalha nao foi acionado quando o xFalhaInversor estava em falha'));

		stMotor.En.xTemInversor		:= FALSE;
		stMotor.En.xFalhaInversor	:= FALSE;
		Partida(stMotor := stMotor);

		//inversor em offline
		stMotor.En.xTemInversor		:= TRUE;
		stMotor.En.xInversorOnline	:= FALSE;
		Partida(stMotor := stMotor);

		AssertEquals_BOOL
			(
				Expected := TRUE,
					Actual := stMotor.Sa.xFalha,
					Message := ('xFalha nao foi acionado quando o xInversorOnline estava em falha'));

		stMotor.En.xTemInversor		:= FALSE;
		stMotor.En.xInversorOnline	:= FALSE;
		Partida(stMotor := stMotor);

		xFaltaSoOsQueTemTempo := TRUE;
	END_IF

	stMotor.En.xLigaAuto					:= TRUE;
	stMotor.En.xContatorLigado				:= FALSE;
	stMotor.Config.rTempoFeedBackContator	:= 1.5;
	Partida(stMotor := stMotor);

	tonFalha(IN := stMotor.Sa.xCmdFwd, PT := REAL_TO_TIME(stMotor.Config.rTempoFeedBackContator * 1000), Q =>, ET =>);

	IF tonFalha.q THEN
		Partida(stMotor := stMotor);

		AssertEquals_BOOL
			(
				Expected := TRUE,
					Actual := stMotor.Sa.xFalha,
					Message := ('xFalha nao foi acionado quando o contato nao veio no tempo esperado'));

		xTerminouTodos := TRUE;
	END_IF

	IF xTerminouTodos THEN
		stMotor.En.xReset		:= TRUE;
		stMotor.En.xLigaAuto	:= FALSE;
		Partida(stMotor := stMotor);
		stMotor.En.xReset := FALSE;

		xTerminouTodos			:= FALSE;
		xFaltaSoOsQueTemTempo	:= FALSE;
		TEST_FINISHED();
	END_IF

END_IF
END_METHOD

METHOD PRIVATE Interlocks
VAR

END_VAR
IF TEST_ORDERED('Interlocks') THEN

	stMotor := stMotorVazio;

	//config inicial da partida
	xLicensaValida5154156 := true;
	Partida(stMotor := stMotor);


	FOR i := 1 TO 4 DO
		stMotor.En.xEmergenciaOK		:= TRUE;
		stMotor.En.xLigaAuto			:= TRUE;
		stMotor.En.xContatorLigado		:= TRUE;
		stMotor.En.xDisjuntorOK			:= TRUE;
		stMotor.En.xAutomaticoManual	:= TRUE;
		stMotor.En.xBloqueado			:= FALSE;
		stMotor.En.xLigaHigienizacao	:= FALSE;
		CASE i OF
			1:
				stMotor.En.xInterLock_1 := TRUE;

			2:
				stMotor.En.xInterLock_2 := TRUE;

			3:
				stMotor.En.xInterLock_3 := TRUE;

			4:
				stMotor.En.xInterLock_4 := TRUE;

		END_CASE

		Partida(stMotor := stMotor);
		Partida(stMotor := stMotor);

		AssertEquals_BOOL
			(
				Expected := TRUE,
					Actual := stMotor.Sa.xLigado,
					Message := CONCAT('xLigado nao estava acionado com interlock', INT_TO_STRING(i)));

		AssertEquals_BOOL
			(
				Expected := FALSE,
					Actual := stMotor.Sa.xCmdFwd,
					Message := CONCAT('xCmdFwd acionado com interlock', INT_TO_STRING(i)));

		AssertEquals_BOOL
			(
				Expected := FALSE,
					Actual := stMotor.Sa.xCmdRev,
					Message := CONCAT('xCmdRev acionado com interlock', INT_TO_STRING(i)));

		AssertEquals_BOOL
			(
				Expected := TRUE,
					Actual := stMotor.Sa.xParadoPorInterlock,
					Message := CONCAT('Nao foi acionado xParadoPorInterlock no interlock', INT_TO_STRING(i)));

		stMotor.En.xInterLock_1	:= FALSE;
		stMotor.En.xInterLock_2	:= FALSE;
		stMotor.En.xInterLock_3	:= FALSE;
		stMotor.En.xInterLock_4	:= FALSE;
		Partida(stMotor := stMotor);
	END_FOR

	TEST_FINISHED();

END_IF
END_METHOD

METHOD PRIVATE ProxPartida
VAR
END_VAR
IF TEST_ORDERED('ProxParida') THEN

	IF NOT xComecou THEN

		stMotor := stMotorVazio;

		//config inicial da partida
		Partida(stMotor := stMotor);

		stMotor.En.xEmergenciaOK		:= true;
		stMotor.En.xContatorLigado		:= TRUE;
		stMotor.En.xDisjuntorOK			:= TRUE;
		stMotor.En.xAutomaticoManual	:= TRUE;
		stMotor.En.xBloqueado			:= FALSE;
		xComecou						:= true;

		Partida(stMotor := stMotor);
		//final ocnfig inicial da partida

	END_IF

	stMotor.Config.rTempoProxMotor	:= 1.5;
	stMotor.En.xLigaAuto			:= TRUE;

	Partida(stMotor := stMotor);

	tonProxPartida(IN := stMotor.Sa.xCmdFwd, PT := REAL_TO_TIME(stMotor.Config.rTempoProxMotor * 1000), Q =>, ET =>);

	IF tonProxPartida.q THEN
		Partida(stMotor := stMotor);

		AssertEquals_BOOL
			(
				Expected := FALSE,
					Actual := stMotor.Sa.xNaoLigaProxMotor,
					Message := 'stMotor.Sa.xNaoLigaProxMotor nao desligou no tempo esperado');

		xTerminouTodos := TRUE;
	END_IF

END_IF

IF xTerminouTodos THEN
	xTerminouTodos			:= FALSE;
	xFaltaSoOsQueTemTempo	:= FALSE;
	xComecou				:= FALSE;
	TEST_FINISHED();
END_IF
END_METHOD

METHOD PRIVATE Reversao
VAR
	iaux : INT;
END_VAR
IF TEST_ORDERED('Reversão') THEN

	CASE EstadoReversao OF
		0:
			stMotor := stMotorVazio;

			//config inicial da partida
			Partida(stMotor := stMotor);

			stMotor.En.xEmergenciaOK		:= TRUE;
			stMotor.En.xLigaAuto			:= TRUE;
			stMotor.En.xContatorLigado		:= TRUE;
			stMotor.En.xDisjuntorOK			:= TRUE;
			stMotor.En.xAutomaticoManual	:= TRUE;
			stMotor.En.xBloqueado			:= FALSE;

			Partida(stMotor := stMotor);
			//final ocnfig inicial da partida
			EstadoReversao := 1;

		1:

			//ve se liga em sentido normal
			stMotor.config.xTemReversao	:= TRUE;
			stMotor.En.xLigaAuto		:= TRUE;
			Partida(stMotor := stMotor);

			AssertEquals_BOOL
				(
					Expected := TRUE,
						Actual := stMotor.Sa.xCmdFwd,
						Message := 'stMotor.Sa.xCmdFwd nao ligou quando deveria em automatico');

			AssertEquals_BOOL
				(
					Expected := FALSE,
						Actual := stMotor.Sa.xCmdRev,
						Message := 'stMotor.Sa.xCmdRev ligou quando nao deveria em automatico');

			EstadoReversao	:= 2;
			xAux			:= FALSE;

		2:

			//ve se liga em sentido normal
			stMotor.config.xTemReversao					:= TRUE;
			stMotor.config.rTempoTrocaSentidoDeMarcha	:= 1.5;
			stMotor.En.xLigaAuto						:= TRUE;
			stMotor.En.xReversoAuto						:= TRUE;
			Partida(stMotor := stMotor);

			IF NOT xAux THEN // olha ver se ele ligou o trocando o sentido
				Partida(stMotor := stMotor);

				AssertEquals_BOOL
					(
						Expected := TRUE,
							Actual := stMotor.Sa.xTrocandoSentido,
							Message := 'stMotor.Sa.xTrocandoSentido nao ligou quando começou a fazer a reverçao em automatico');

				AssertEquals_BOOL
					(
						Expected := TRUE,
							Actual := stMotor.Sa.xLigado,
							Message := 'stMotor.Sa.xLigado nao ficou ligado quando começou a fazer a reverçao em automatico');

				xAux := TRUE;
			END_IF

			tonReversao(IN := stMotor.En.xLigaAuto, PT := REAL_TO_TIME(stMotor.config.rTempoTrocaSentidoDeMarcha * 1000), Q =>, ET =>);

			IF tonReversao.q THEN
				Partida(stMotor := stMotor);

				AssertEquals_BOOL
					(
						Expected := FALSE,
							Actual := stMotor.Sa.xCmdFwd,
							Message := 'stMotor.Sa.xCmdFwd ligou quando ja deveria ter termiando de fazer a reversao em automatico');

				AssertEquals_BOOL
					(
						Expected := TRUE,
							Actual := stMotor.Sa.xCmdRev,
							Message := 'stMotor.Sa.xCmdRev nao ligou apos ter feito a reversao em automatico');

				EstadoReversao := 3;
				tonReversao(IN := FALSE, PT :=, Q =>, ET =>);
			END_IF

		3:
			stMotor.En.xReversoAuto	:= FALSE;
			stMotor.En.xLigaAuto	:= FALSE;
			Partida(stMotor := stMotor);
			tonReversao(IN := TRUE, PT := REAL_TO_TIME(stMotor.config.rTempoTrocaSentidoDeMarcha * 1000), Q =>, ET =>);

			IF tonReversao.q THEN
				tonReversao(IN := FALSE, PT :=, Q =>, ET =>);
				EstadoReversao := 4;
			END_IF

		4:

			stMotor.En.xAutomaticoManual := FALSE;
			Partida(stMotor := stMotor);

			//ve se liga em sentido normal
			stMotor.config.xTemReversao	:= TRUE;
			stMotor.En.xLigaManu		:= TRUE;
			Partida(stMotor := stMotor);

			AssertEquals_BOOL
				(
					Expected := TRUE,
						Actual := stMotor.Sa.xCmdFwd,
						Message := 'stMotor.Sa.xCmdFwd nao ligou quando deveria em manual');

			AssertEquals_BOOL
				(
					Expected := FALSE,
						Actual := stMotor.Sa.xCmdRev,
						Message := 'stMotor.Sa.xCmdRev ligou quando nao deveria em manual');

			EstadoReversao	:= 5;
			xAux			:= FALSE;

		5:
			//ve se liga em sentido normal
			stMotor.config.xTemReversao					:= TRUE;
			stMotor.config.rTempoTrocaSentidoDeMarcha	:= 1.5;
			stMotor.En.xLigaManu						:= TRUE;
			stMotor.En.xReversoManu						:= TRUE;
			Partida(stMotor := stMotor);

			IF NOT xAux THEN // olha ver se ele ligou o trocando o sentido
				Partida(stMotor := stMotor);

				AssertEquals_BOOL
					(
						Expected := TRUE,
							Actual := stMotor.Sa.xTrocandoSentido,
							Message := 'stMotor.Sa.xTrocandoSentido nao ligou quando começou a fazer a reverçao em manual');

				AssertEquals_BOOL
					(
						Expected := TRUE,
							Actual := stMotor.Sa.xLigado,
							Message := 'stMotor.Sa.xLigado nao ficou ligado quando começou a fazer a reverçao em manual');

				xAux := TRUE;
			END_IF

			tonReversao(IN := stMotor.En.xLigaManu, PT := REAL_TO_TIME(stMotor.config.rTempoTrocaSentidoDeMarcha * 1000), Q =>, ET =>);

			IF tonReversao.q THEN
				Partida(stMotor := stMotor);

				AssertEquals_BOOL
					(
						Expected := FALSE,
							Actual := stMotor.Sa.xCmdFwd,
							Message := 'stMotor.Sa.xCmdFwd ligou quando ja deveria ter termiando de fazer a reversao em manual');

				AssertEquals_BOOL
					(
						Expected := TRUE,
							Actual := stMotor.Sa.xCmdRev,
							Message := 'stMotor.Sa.xCmdRev nao ligou apos ter feito a reversao em manual');

				tonReversao(IN := FALSE, PT :=, Q =>, ET =>);
				EstadoReversao := 6;
			END_IF

		6:
			stMotor.En.xReversoManu	:= TRUE;
			stMotor.En.xLigaManu	:= FALSE;
			stMotor.En.xReversoAuto	:= TRUE;
			stMotor.En.xLigaauto	:= FALSE;
			Partida(stMotor := stMotor);
			tonReversao(IN := TRUE, PT := REAL_TO_TIME(stMotor.config.rTempoTrocaSentidoDeMarcha * 1000), Q =>, ET =>);

			IF tonReversao.q THEN
				tonReversao(IN := FALSE, PT :=, Q =>, ET =>);
				EstadoReversao := 7;
			END_IF

		7:
			stMotor.En.xReversoManu			:= TRUE;
			stMotor.En.xLigaManu			:= TRUE;
			stMotor.En.xReversoAuto			:= TRUE;
			stMotor.En.xLigaauto			:= TRUE;
			stMotor.En.xAutomaticoManual	:= FALSE;
			Partida(stMotor := stMotor);

			stMotor.En.xReversoManu			:= TRUE;
			stMotor.En.xLigaManu			:= TRUE;
			stMotor.En.xReversoAuto			:= TRUE;
			stMotor.En.xLigaauto			:= TRUE;
			stMotor.En.xAutomaticoManual	:= TRUE;
			Partida(stMotor := stMotor);

			AssertEquals_BOOL
				(
					Expected := TRUE,
						Actual := stMotor.Sa.xCmdRev,
						Message := 'Apos fazer troca de manual pra automatico ele nao manteve o comando de marcha reverso, mesmo sendo automatico e manual pro mesmo lado');

			EstadoReversao := 8;

		8:
			stMotor.En.xReversoManu	:= FALSE;
			stMotor.En.xLigaManu	:= FALSE;
			stMotor.En.xReversoAuto	:= FALSE;
			stMotor.En.xLigaauto	:= FALSE;
			Partida(stMotor := stMotor);
			tonReversao(IN := TRUE, PT := REAL_TO_TIME(stMotor.config.rTempoTrocaSentidoDeMarcha * 1000), Q =>, ET =>);

			IF tonReversao.q THEN
				tonReversao(IN := FALSE, PT :=, Q =>, ET =>);
				EstadoReversao := 9;
			END_IF

		9:
			stMotor.En.xReversoManu			:= FALSE;
			stMotor.En.xLigaManu			:= TRUE;
			stMotor.En.xReversoAuto			:= FALSE;
			stMotor.En.xLigaauto			:= TRUE;
			stMotor.En.xAutomaticoManual	:= FALSE;
			Partida(stMotor := stMotor);

			stMotor.En.xReversoManu			:= FALSE;
			stMotor.En.xLigaManu			:= TRUE;
			stMotor.En.xReversoAuto			:= FALSE;
			stMotor.En.xLigaauto			:= TRUE;
			stMotor.En.xAutomaticoManual	:= TRUE;
			Partida(stMotor := stMotor);

			AssertEquals_BOOL
				(
					Expected := TRUE,
						Actual := stMotor.Sa.xCmdFwd,
						Message :=
						'Apos fazer troca de manual pra automatico ele nao manteve o comando de marcha, mesmo sendo automatico e manual pro mesmo lado');

			EstadoReversao := 10;

		10:
			stMotor.En.xReversoManu	:= FALSE;
			stMotor.En.xLigaManu	:= FALSE;
			stMotor.En.xReversoAuto	:= FALSE;
			stMotor.En.xLigaauto	:= FALSE;
			Partida(stMotor := stMotor);
			tonReversao(IN := TRUE, PT := REAL_TO_TIME(stMotor.config.rTempoTrocaSentidoDeMarcha * 1000), Q =>, ET =>);

			IF tonReversao.q THEN
				tonReversao(IN := FALSE, PT :=, Q =>, ET =>);
				EstadoReversao := 11;
			END_IF

		11:
			IF NOT xAux THEN
				stMotor.En.xReversoManu			:= FALSE;
				stMotor.En.xLigaManu			:= TRUE;
				stMotor.En.xReversoAuto			:= FALSE;
				stMotor.En.xLigaauto			:= FALSE;
				stMotor.En.xAutomaticoManual	:= FALSE;
				Partida(stMotor := stMotor);
				xAux := TRUE;
			END_IF

			stMotor.En.xReversoManu			:= FALSE;
			stMotor.En.xLigaManu			:= FALSE;
			stMotor.En.xReversoAuto			:= FALSE;
			stMotor.En.xLigaauto			:= TRUE;
			stMotor.En.xAutomaticoManual	:= TRUE;
			Partida(stMotor := stMotor);

			tonReversao(IN := TRUE, PT := REAL_TO_TIME(stMotor.config.rTempoTrocaSentidoDeMarcha * 1000), Q =>, ET =>);

			IF tonReversao.q THEN
				tonReversao(IN := FALSE, PT :=, Q =>, ET =>);
				EstadoReversao	:= 100;
				xAux			:= FALSE;
			END_IF

		100:
			TEST_FINISHED();

	END_CASE
END_IF
END_METHOD

METHOD PRIVATE Velocidade
VAR
	iaux : INT;
END_VAR
IF TEST_ORDERED('Velocidade') THEN

	stMotor := stMotorVazio;

	//config inicial da partida
	Partida(stMotor := stMotor);

	stMotor.En.xEmergenciaOK		:= TRUE;
	stMotor.En.xLigaAuto			:= TRUE;
	stMotor.En.xContatorLigado		:= TRUE;
	stMotor.En.xDisjuntorOK			:= TRUE;
	stMotor.En.xAutomaticoManual	:= FALSE;
	stMotor.En.xBloqueado			:= FALSE;

	xLicensaValida5154156 := true;

	//velo em manual
	Partida(stMotor := stMotor);
	Partida(stMotor := stMotor);
	stMotor.Config.rSetPoinManu := 100;
	Partida(stMotor := stMotor);
	iaux := TO_INT(stMotor.Config.rSetPoinManu); 
	
	AssertEquals
		(
			Expected := iaux,
				Actual := stMotor.Sa.iVelocidade,
				Message := 'Velocidade em manual nao funcionou');

	//velo base em automatico
	stMotor.En.xAutomaticoManual	:= TRUE;
	Partida(stMotor := stMotor);
	Partida(stMotor := stMotor);
	stMotor.Config.rSetPoinAuto		:= 100;
	Partida(stMotor := stMotor);
	iaux := TO_INT(stMotor.Config.rSetPoinAuto);

	AssertEquals
		(
			Expected := iaux,
				Actual := stMotor.Sa.iVelocidade,
				Message := 'Velocidade sem comissionamento em automatico nao funcionou');

	//velo em % comissionada em automatico		
	stMotor.En.xAutomaticoManual				:= TRUE;
	stMotor.Config.rVeloEmPorcentagem_VeloMax	:= 1500;
	stMotor.Config.xComissionado_Corrente		:= TRUE;
	stMotor.Config.xComissionado_Sentido		:= TRUE;
	stMotor.Config.xComissionado_Velo			:= TRUE;
	stMotor.Config.xVeloEmPorcentagem			:= TRUE;
	Partida(stMotor := stMotor);
	Partida(stMotor := stMotor);
	stMotor.Config.rSetPoinAuto					:= 100;
	Partida(stMotor := stMotor);
	iaux := 1500;

	AssertEquals
		(
			Expected := iaux,
				Actual := stMotor.Sa.iVelocidade,
				Message := 'Velocidade comissionada em % nao funcionou');

	//velo p/min comissionada em automatico		
	stMotor.En.xAutomaticoManual				:= TRUE;
	stMotor.Config.rVeloEmMetroPMin_Conversao	:= 10;
	stMotor.Config.xComissionado_Corrente		:= TRUE;
	stMotor.Config.xComissionado_Sentido		:= TRUE;
	stMotor.Config.xComissionado_Velo			:= TRUE;
	stMotor.Config.xVeloEmPorcentagem			:= FALSE;
	stMotor.Config.xVeloEmMetroPMin				:= TRUE;
	Partida(stMotor := stMotor);
	Partida(stMotor := stMotor);
	stMotor.Config.rSetPoinAuto					:= 5;
	Partida(stMotor := stMotor);
	iaux := 900;

	AssertEquals
		(
			Expected := iaux,
				Actual := stMotor.Sa.iVelocidade,
				Message := 'Velocidade comissionada em p/min nao funcionou');

	//sentido comissionado		
	stMotor.En.xAutomaticoManual				:= TRUE;
	stMotor.Config.rVeloEmMetroPMin_Conversao	:= 10;
	stMotor.Config.xComissionado_Corrente		:= TRUE;
	stMotor.Config.xComissionado_Sentido		:= TRUE;
	stMotor.Config.xComissionado_Velo			:= TRUE;
	stMotor.Config.xVeloEmMetroPMin				:= TRUE;
	stMotor.Config.xInverteSentido				:= TRUE;
	Partida(stMotor := stMotor);
	Partida(stMotor := stMotor);
	stMotor.Config.rSetPoinAuto					:= 5;
	Partida(stMotor := stMotor);
	iaux := -900;

	AssertEquals
		(
			Expected := iaux,
				Actual := stMotor.Sa.iVelocidade,
				Message := 'Velocidade invertida nao funcionou em automatico');

	//velo em manual
	stMotor.En.xAutomaticoManual	:= FALSE;
	Partida(stMotor := stMotor);
	Partida(stMotor := stMotor);
	stMotor.Config.rSetPoinManu		:= 100;
	Partida(stMotor := stMotor);
	iAux := -18000;

	AssertEquals
		(
			Expected := iAux,
				Actual := stMotor.Sa.iVelocidade,
				Message := 'Velocidade invertida nao funcionou em manual');

	TEST_FINISHED();

END_IF
END_METHOD

END_FUNCTION_BLOCK

// POUs/Partida/FB_Partida
{attribute 'hide_all_locals'}
FUNCTION_BLOCK FB_Partida
VAR_IN_OUT
	stMotor : st_Partida;
END_VAR
VAR_INPUT
	xEmergenciaOK		: BOOL;	(*Sinal de Emergência*)
	xFaltaDeFaseOk 		: BOOL; // Se o falta de fase esta OK
	xTemContatora		: BOOL; // pra considerar ou nao a contatora no programa
	xContatorLigado		: BOOL;	(*Status da contatora ou do drive de que o motor partiu*)
	xByPassContator		: BOOL;	//Sinal de by pass do contato da contatora
	xTemDisjuntor		: BOOL; // pra considerar ou nao o disjuntor no programa
	xDisjuntorOK		: BOOL;	(*Status do disjuntor motor*)
	xByPassDisjuntor	: BOOL;	//Sinal de by pass do contato do disjuntor
	xBloqueado			: BOOL;	//Sinal de Bloqueio
	iSenhaBloqueio		: INT;	//Senha de bloqueio
	iSenhaAtual			: INT;	// Senha que aparece no HMI
	xAutomaticoManual	: BOOL;	// se automatico = true se manual = false
	xLigaHigienizacao	: BOOL; // Define que a esteira esta em modo de Higienização
	xHabilitaHigienizacao: BOOL; // Se tiver em true quando tiver xLigaHigienizacao ele vai ligar a esteira em 10% da velo
	rSetPoinAuto		: REAL;	// velocidadde que sera mandada para o bloco de comunicação
	xUsaVeloAuto2		: BOOL; // Usa a segunda velo em automatico
	rSetPoinAuto2		: REAL;	// velocidadde que sera mandada para o bloco de comunicação
	xReversoAuto		: BOOL;	// comando para ligar reverso o motor
	xLigaAuto			: BOOL;	// liga inversor em automatico
	rSetPoinManu		: real;	// velocidadde que sera mandada para o bloco de comunicação
	xReversoManu		: BOOL;	// Comando para ligar ele reverso
	xLigaManu			: BOOL;	// liga inversor em manual
	xLigaManu3S			: BOOL;	// Liga por 3 segundos em manual(Para comissionamento)
	xReset				: BOOL;	(*Sinal para resetar as falhas*)
	xResetaNumeroDeReset: BOOL;
	xResetRegistros		: BOOL;	(*Sinal apra resetar os contadores e registradores*)

	//Bloqueios
	xInterLock_1	: BOOL;		// sinal para bloquear a partida
	sInterLock_1	: STRING;	// porque o bloqueio 1
	xInterLock_2	: BOOL;		// sinal para bloquear a partida
	sInterLock_2	: STRING;	// porque o bloqueio 1
	xInterLock_3	: BOOL;		// sinal para bloquear a partida
	sInterLock_3	: STRING;	// porque o bloqueio 1
	xInterLock_4	: BOOL;		// sinal para bloquear a partida
	sInterLock_4	: STRING;	// porque o bloqueio 1

	//Inversor/comunicacao caso tenha
	xTemInversor	: BOOL;	// define se o bloco considera ou nao uma conexao
	xTemTeSysU		: BOOL;
	xInversorOnline	: BOOL;	// se etiver online
	xFalhaInversor	: BOOL;	// se o inversor tiver qualquer outra falha que nao seja perda de conexao
	xBypassRede		: BOOL;	// para caso tenha problema na rede ele poder operar sem ela
	xLocal			: BOOL; // se o inversor esta em modo local ou remoto
	xResetBlocoComunicacao : BOOL; //o reset do bloco vempor aqui, ai nao bate na contagem do reset
	
	xTemContatoInversorOK 		: BOOL; // se tem contato de OK do inversor
	xBypassContatoInversorOK 	: BOOL; // bypass do contato de OK do inversor
	xContatoInversorOK 			: BOOL; // contato de OK do inversor
	
	stHoraAgora : TIMESTRUCT; // struct de hora para o horimetro

	xFazendoComissionamento : BOOL; // quando tiver fazendo o comissionamento ela fica true

	xBypassFreio	: BOOL;
	xFreioOK		: BOOL;
	
	xBypassContatoFalhaSoft : BOOL;
	xContatoFalhaSoft : BOOL;
	xBypassContatoRunSoft : BOOL;
	xContatoRodandoSoft : BOOL;
	xSoftOnline : BOOL;
	xSoftEmFalhaCOM : BOOL;
	xBypassSoftEmFalhaCOM : BOOL;
	
	
	rPorcentagemHigienizacao : REAL;
	
	xECO : BOOL;

END_VAR
VAR_OUTPUT
	xLigado				: BOOL;	// sinal que o motor ta ligado, apesar de ele ter parado para fazer a reversao ou pelos interlocks
	xCmdFwd				: BOOL;	(*Liga Motor pra frente*)
	xCmdRev				: BOOL;	(*Liga Motor pra Tras*)
	xTrocandoSentido	: BOOL;	// sinal de que ele ta trocando o sentido de giro e por isso ele ta parado
	xParadoPorInterlock	: BOOL;	// se ele parar por algum interlock ele mostra aqui
	iVelocidade			: INT;	// velocidade para bloco de comunicação
	iStsMotor			: INT;
	xResetParaInversor	: BOOL;	// sinal para o drive dar reset
	xFalha				: BOOL;	//Partida em falha
	sStatus 			: STRING;// Status da partida
	xFalhaContatora 	: BOOL; //Sinal de falha da contatora para a IHM
	iDisjDesarm			: INT;	(*Contagem do numero de desarmes do disjuntor*)
	iPartidas			: INT;	(*Contagem do numero de partidas com sucesso do bloco*)
	iFalhaPartida		: INT;	(*Contagem do numero de falhas na partida do bloco*)
	// dados vindo do inversor, coloquei aqui para facilitar a visualização
	rVoltagemEntrada	: REAL;
	rTorque				: REAL;
	rTemperaturaInver	: REAL;
	rTemperaturaMotor	: REAL;
	rCorrente			: REAL;
	rVelocidadeRPM		: REAL;
	rVelocidadeHz		: REAL;
	sUltimoErro			: STRING;
	sStatusConexao		: STRING;

	//Conversao de velo em automatico

	xComissionado_Sentido	: BOOL;
	xInverteSentido			: BOOL; // bit pra inverrter o sentido do inversor

	xComissionado_Velo : BOOL;

	xVeloEmPorcentagem			: BOOL;	// usa o valor de 0-100% para controle da velo
	rVeloEmPorcentagem_VeloMax	: REAL;	// velo que representa 100%

	xVeloEmMetroPMin			: BOOL;	// usa a conversao para calcular a velocidade usada
	rVeloEmMetroPMin_Conversao	: REAL;	// valor em m/Min em 1000 RPM

	xComissionado_Corrente	: BOOL;
	rCorrente_Comissionada	: REAL;

	xTudoComissionado : BOOL;
	
	xFalhaPartidaSoft : BOOL;

	///Horimetro

	tHorimetro	: TIME;
	sHorimetro	: STRING;

	xNaoLigaProxMotor : BOOL;

	// nome do motor e função para IHM
	sNome_Funcao : STRING;

END_VAR
VAR
	TON_Partida				: TON;
	rtFalhanaPartida		: R_TRIG;
	rtSucessonaPartida		: R_TRIG;
	rtDisjuntorDesarmado	: R_TRIG;
	Ultima_stMotor			: st_Partida;
	rtVoltouOnline			: R_TRIG;
	tonReset				: TON; // ton reset pra ele nao ficar preso
	xTavaEmEmergencia		: BOOL;
	rtTavaEmEmergencia		: R_TRIG;
	rtVoltaEmergencia		: R_TRIG;
	Ton3Segundos			: TON;
	Ton3SegundosOff			: TON;
	xOffTempoOK				: BOOL;
	systime					: GETSYSTEMTIME;
	currentTime				: T_FILETIME;
	dtAux					: DT;
	timeStructAux			: TIMESTRUCT;
	wDiaAnterior			: WORD;

	tonLigaProxMotor : TON;

	btTrocouSentidoRotAuto		: B_TRIG;
	btTrocouSentidoRotManu		: B_TRIG;
	btTrocouManualAutomatico	: B_TRIG;
	tpTrocaSentidoDeRotacao		: TP;

	ftManual : F_TRIG;

	rtBloqueiou		: R_TRIG;
	rtDesbloquiou	: f_TRIG;

	xFirstScan		: BOOL := TRUE;

	i				: INT;
	wSegAnterior	: WORD;
	whoraAnterior	: WORD;
	kpiVazio		: st_KPIPartida;
	
	TON_Soft		: TON;
	rAux : REAL;
	
	rtSaiComissionamento : R_TRIG;
	
	rtReset : R_TRIG;
	tonResetFalha : TON;
	
	fbHorimetro : FB_HorimetroTime_Otimizado;
	
	iaux : INT;
	
	rtLigou : b_TRIG;
	rtfalha : R_TRIG;
	rtEmergencia : R_TRIG;
	rtInterlock : R_TRIG;
	
	//OEE
	rAux1 : REAL;
	rAux2 : REAL;
	
	udiLigado : UDINT;
	udiFalha : UDINT;
	udiEmergencia : UDINT;
	udiinterlock : UDINT;
	
	udiDisponibilidade 	: UDINT;
	udiPerformace 		: UDINT;
	udiQualidade	 	: UDINT;
	
	tTempoComxLigaAuto 	: TIME;
	tXligaEEmergencia 	: TIME;
	tXligaEInterlock 	: TIME;
	tXligaEFalha 		: TIME;
	
	
	
END_VAR

//========================================================================
//FB de partida da TEKNIKE
//feito por Tiago Bortolini Cunico em 31/10/2021
//foi usado codigo feito pelo Ricardo Gajardo tambem
//A ideia é que esta partida funciona como a partida direta, porem os 
//blocos de comunicação recebem a estrutura dessa partida e nela utilizam
//para o controle do inversor
//========================================================================
IF xLicensaValida5154156 THEN
	
	
	IF xFirstScan THEN
		FirstScan();
	END_IF
	
	AjustaEntradaST();
	
	ControleBloqueio();
	ControleReset();
	
	tonReset(IN := xReset OR xResetBlocoComunicacao, PT := T#500MS, Q =>, ET =>);
	
	IF tonReset.q THEN
		xReset := FALSE;
		xResetBlocoComunicacao := FALSE;
	END_IF
	
	IF xReset OR xResetBlocoComunicacao THEN
		xFalha					:= FALSE;
		xFazendoComissionamento	:= FALSE;
	END_IF
	
	
	IF NOT xFazendoComissionamento THEN
		ControleDaPartida();
		ControleVelocidade();
	ELSE
		EmComissionamento();
	END_IF
	
	SegurancaReversao();
	
	Falhas();
	
	Status();
	
	Contagem();
	
	ProxMotor();
	
	Horimetro();
	
	KPI();
	
	AlarmesIHM();
	
	AjustaSaida();
	
	xFirstScan := FALSE;

ELSE
	ValidaLicensa();
END_IF

ACTION AjustaEntradaST:

//Esse é diferente por que tem que vim o valor retentivo primeiro
//do st pro fb
IF stMotor.Config.rSetPoinAuto <> Ultima_stMotor.Config.rSetPoinAuto THEN
	rSetPoinAuto := stMotor.Config.rSetPoinAuto;
END_IF

IF stMotor.Config.rSetPoinManu <> Ultima_stMotor.Config.rSetPoinManu THEN
	rSetPoinManu := stMotor.Config.rSetPoinManu;
END_IF

IF stMotor.Config.xByPassContator <> Ultima_stMotor.Config.xByPassContator THEN
	xByPassContator := stMotor.Config.xByPassContator;
END_IF

IF stMotor.Config.xByPassDisjuntor <> Ultima_stMotor.Config.xByPassDisjuntor THEN
	xByPassDisjuntor := stMotor.Config.xByPassDisjuntor;
END_IF

IF stMotor.Config.xBypassRede <> Ultima_stMotor.Config.xBypassRede THEN
	xBypassRede := stMotor.Config.xBypassRede;
END_IF

IF stMotor.Config.xBypassFreio <> Ultima_stMotor.Config.xBypassFreio THEN
	xBypassFreio := stMotor.Config.xBypassFreio;
END_IF

IF stMotor.Config.xTemContatoInversorOK <> Ultima_stMotor.Config.xTemContatoInversorOK THEN
	xTemContatoInversorOK := stMotor.Config.xTemContatoInversorOK;
END_IF

IF stMotor.Config.xBypassContatoRunSoft <> Ultima_stMotor.Config.xBypassContatoRunSoft THEN
	xBypassContatoRunSoft := stMotor.Config.xBypassContatoRunSoft;
END_IF

IF stMotor.Config.xBypassContatoFalhaSoft <> Ultima_stMotor.Config.xBypassContatoFalhaSoft THEN
	xBypassContatoFalhaSoft := stMotor.Config.xBypassContatoFalhaSoft;
END_IF

IF stMotor.Config.xBypassSoftEmFalhaCOM <> Ultima_stMotor.Config.xBypassSoftEmFalhaCOM THEN
	xBypassSoftEmFalhaCOM := stMotor.Config.xBypassSoftEmFalhaCOM;
END_IF

IF stMotor.Config.rSetPoinAuto2 <> Ultima_stMotor.Config.rSetPoinAuto2 THEN
	rSetPoinAuto2 := stMotor.Config.rSetPoinAuto2;
END_IF

IF stMotor.Config.xHabilitaHigienizacao <> Ultima_stMotor.Config.xHabilitaHigienizacao THEN
	xHabilitaHigienizacao := stMotor.Config.xHabilitaHigienizacao;
END_IF

IF stMotor.Config.rPorcentagemHigienizacao <> Ultima_stMotor.Config.rPorcentagemHigienizacao THEN
	rPorcentagemHigienizacao := stMotor.Config.rPorcentagemHigienizacao;
END_IF

IF xBypassContatoInversorOK <> Ultima_stMotor.Config.xBypassContatoInversorOK THEN
	stMotor.Config.xBypassContatoInversorOK := xBypassContatoInversorOK;
END_IF

IF xTemContatora <> Ultima_stMotor.Config.xTemContatora THEN
	stMotor.Config.xTemContatora := xTemContatora;
END_IF

IF xTemDisjuntor <> Ultima_stMotor.Config.xTemDisjuntor THEN
	stMotor.Config.xTemDisjuntor := xTemDisjuntor;
END_IF


//Do ST pro FB	
IF rSetPoinAuto <> Ultima_stMotor.Config.rSetPoinAuto THEN
	stMotor.Config.rSetPoinAuto := rSetPoinAuto;
END_IF

IF rSetPoinManu <> Ultima_stMotor.Config.rSetPoinManu THEN
	stMotor.Config.rSetPoinManu := rSetPoinManu;
END_IF

IF xByPassContator <> Ultima_stMotor.Config.xByPassContator THEN
	stMotor.Config.xByPassContator := xByPassContator;
END_IF

IF xByPassDisjuntor <> Ultima_stMotor.Config.xByPassDisjuntor THEN
	stMotor.Config.xByPassDisjuntor := xByPassDisjuntor;
END_IF

IF xBypassRede <> Ultima_stMotor.Config.xBypassRede THEN
	stMotor.Config.xBypassRede := xBypassRede;
END_IF

IF stMotor.Config.xBypassFreio <> xBypassFreio THEN
	stMotor.Config.xBypassFreio := xBypassFreio;
END_IF

IF stMotor.Config.xTemContatoInversorOK <> xTemContatoInversorOK THEN
	stMotor.Config.xTemContatoInversorOK := xTemContatoInversorOK;
END_IF

IF stMotor.Config.xBypassContatoRunSoft <> xBypassContatoRunSoft THEN
	 stMotor.Config.xBypassContatoRunSoft := xBypassContatoRunSoft;
END_IF

IF stMotor.Config.xBypassContatoFalhaSoft <> xBypassContatoFalhaSoft THEN
	 stMotor.Config.xBypassContatoFalhaSoft := xBypassContatoFalhaSoft;
END_IF

IF stMotor.Config.xBypassSoftEmFalhaCOM <> xBypassSoftEmFalhaCOM THEN
	 stMotor.Config.xBypassSoftEmFalhaCOM := xBypassSoftEmFalhaCOM;
END_IF

IF stMotor.Config.rSetPoinAuto2 <> rSetPoinAuto2 THEN
	 stMotor.Config.rSetPoinAuto2 := rSetPoinAuto2;
END_IF

IF stMotor.Config.xHabilitaHigienizacao <> xHabilitaHigienizacao THEN
	 stMotor.Config.xHabilitaHigienizacao := xHabilitaHigienizacao;
END_IF

IF stMotor.Config.rPorcentagemHigienizacao <> rPorcentagemHigienizacao THEN
	 stMotor.Config.rPorcentagemHigienizacao := rPorcentagemHigienizacao;
END_IF
	
IF stMotor.Config.xBypassContatoInversorOK <> Ultima_stMotor.Config.xBypassContatoInversorOK THEN
	xBypassContatoInversorOK := stMotor.Config.xBypassContatoInversorOK;
END_IF
	
IF stMotor.Config.xTemContatora <> Ultima_stMotor.Config.xTemContatora THEN
	xTemContatora := stMotor.Config.xTemContatora;
END_IF
	
IF stMotor.Config.xTemDisjuntor <> Ultima_stMotor.Config.xTemDisjuntor THEN
	xTemDisjuntor := stMotor.Config.xTemDisjuntor;
END_IF



////////////////// OS NAO CONFIG PRA BAIXO



// do fb pro st
IF NOT xFirstScan THEN
	
	IF xEmergenciaOK <> Ultima_stMotor.En.xEmergenciaOK THEN
		stMotor.En.xEmergenciaOK := xEmergenciaOK;
	END_IF
	
	IF xContatorLigado <> Ultima_stMotor.En.xContatorLigado THEN
		stMotor.En.xContatorLigado := xContatorLigado;
	END_IF
	
	IF xDisjuntorOK <> Ultima_stMotor.En.xDisjuntorOK THEN
		stMotor.En.xDisjuntorOK := xDisjuntorOK;
	END_IF
	
	IF xAutomaticoManual <> Ultima_stMotor.En.xAutomaticoManual THEN
		stMotor.En.xAutomaticoManual := xAutomaticoManual;
	END_IF
	
	IF xBloqueado <> Ultima_stMotor.En.xBloqueado THEN
		stMotor.En.xBloqueado := xBloqueado;
	END_IF
	
	IF iSenhaAtual <> Ultima_stMotor.En.iSenhaAtual THEN
		stMotor.En.iSenhaAtual := iSenhaAtual;
	END_IF
	
	IF iSenhaBloqueio <> Ultima_stMotor.En.iSenhaBloqueio THEN
		stMotor.En.iSenhaBloqueio := iSenhaBloqueio;
	END_IF
	
	IF xReversoAuto <> Ultima_stMotor.En.xReversoAuto THEN
		stMotor.En.xReversoAuto := xReversoAuto;
	END_IF
	
	IF xLigaAuto <> Ultima_stMotor.En.xLigaAuto THEN
		stMotor.En.xLigaAuto := xLigaAuto;
	END_IF
	
	IF xReversoManu <> Ultima_stMotor.En.xReversoManu THEN
		stMotor.En.xReversoManu := xReversoManu;
	END_IF
	
	IF xLigaManu <> Ultima_stMotor.En.xLigaManu THEN
		stMotor.En.xLigaManu := xLigaManu;
	END_IF
	
	IF xLigaManu3S <> Ultima_stMotor.En.xLigaManu3S THEN
		stMotor.En.xLigaManu3S := xLigaManu3S;
	END_IF
	
	IF xReset <> Ultima_stMotor.En.xReset THEN
		stMotor.En.xReset := xReset;
	END_IF
	
	IF xResetRegistros <> Ultima_stMotor.En.xResetRegistros THEN
		stMotor.En.xResetRegistros := xResetRegistros;
	END_IF
	
	IF xInterLock_1 <> Ultima_stMotor.En.xInterLock_1 THEN
		stMotor.En.xInterLock_1 := xInterLock_1;
	END_IF
	
	IF sInterLock_1 <> Ultima_stMotor.En.sInterLock_1 THEN
		stMotor.En.sInterLock_1 := sInterLock_1;
	END_IF
	
	IF xInterLock_2 <> Ultima_stMotor.En.xInterLock_2 THEN
		stMotor.En.xInterLock_2 := xInterLock_2;
	END_IF
	
	IF sInterLock_2 <> Ultima_stMotor.En.sInterLock_2 THEN
		stMotor.En.sInterLock_2 := sInterLock_2;
	END_IF
	
	IF xInterLock_3 <> Ultima_stMotor.En.xInterLock_3 THEN
		stMotor.En.xInterLock_3 := xInterLock_3;
	END_IF
	
	IF sInterLock_3 <> Ultima_stMotor.En.sInterLock_3 THEN
		stMotor.En.sInterLock_3 := sInterLock_3;
	END_IF
	
	IF xInterLock_4 <> Ultima_stMotor.En.xInterLock_4 THEN
		stMotor.En.xInterLock_4 := xInterLock_4;
	END_IF
	
	IF sInterLock_4 <> Ultima_stMotor.En.sInterLock_4 THEN
		stMotor.En.sInterLock_4 := sInterLock_4;
	END_IF
	
	IF xTemInversor <> Ultima_stMotor.En.xTemInversor THEN
		stMotor.En.xTemInversor := xTemInversor;
	END_IF
	
	IF xTemTeSysU <> Ultima_stMotor.En.xTemTeSysU THEN
		stMotor.En.xTemTeSysU := xTemTeSysU;
	END_IF
	
	IF xInversorOnline <> Ultima_stMotor.En.xInversorOnline THEN
		stMotor.En.xInversorOnline := xInversorOnline;
	END_IF
	
	IF xFalhaInversor <> Ultima_stMotor.En.xFalhaInversor THEN
		stMotor.En.xFalhaInversor := xFalhaInversor;
	END_IF
	
	IF stHoraAgora.wMilliseconds <> Ultima_stMotor.En.stHoraAgora.wMilliseconds THEN
		stMotor.En.stHoraAgora := stHoraAgora;
	END_IF
	
	IF xFazendoComissionamento <> Ultima_stMotor.En.xFazendoComissionamento THEN
		stMotor.En.xFazendoComissionamento := xFazendoComissionamento;
	END_IF
	
	IF xFreioOK <> Ultima_stMotor.En.xFreioOK THEN
		stMotor.En.xFreioOK := xFreioOK;
	END_IF
	
	IF xContatoInversorOK <> Ultima_stMotor.En.xContatoInversorOK THEN
		stMotor.En.xContatoInversorOK := xContatoInversorOK;
	END_IF
	
	IF xContatoFalhaSoft <> Ultima_stMotor.En.xContatoFalhaSoft THEN
		stMotor.En.xContatoFalhaSoft := xContatoFalhaSoft;
	END_IF
	
	IF xContatoRodandoSoft <> Ultima_stMotor.En.xContatoRodandoSoft THEN
		stMotor.En.xContatoRodandoSoft := xContatoRodandoSoft;
	END_IF
	
	IF xSoftOnline <> Ultima_stMotor.En.xSoftOnline THEN
		stMotor.En.xSoftOnline := xSoftOnline;
	END_IF
	
	IF xUsaVeloAuto2 <> Ultima_stMotor.En.xUsaVeloAuto2 THEN
		stMotor.En.xUsaVeloAuto2 := xUsaVeloAuto2;
	END_IF
	
	IF xLigaHigienizacao <> Ultima_stMotor.En.xLigaHigienizacao THEN
		stMotor.En.xLigaHigienizacao := xLigaHigienizacao;
	END_IF
	
	IF xResetaNumeroDeReset <> Ultima_stMotor.En.xResetaNumeroDeReset THEN
		stMotor.En.xResetaNumeroDeReset := xResetaNumeroDeReset;
	END_IF
		
	IF xLocal <> Ultima_stMotor.En.xLocal THEN
		stMotor.En.xLocal := xLocal;
	END_IF
		
	IF xContatoInversorOK <> Ultima_stMotor.En.xContatoInversorOK THEN
		stMotor.En.xContatoInversorOK := xContatoInversorOK;
	END_IF
		
	IF xECO <> Ultima_stMotor.En.xECO THEN
		stMotor.En.xECO := xECO;
	END_IF
		
	IF xResetBlocoComunicacao <> Ultima_stMotor.En.xResetBlocoComunicacao THEN
		stMotor.En.xResetBlocoComunicacao := xResetBlocoComunicacao;
	END_IF
		
	IF xSoftEmFalhaCOM <> Ultima_stMotor.En.xSoftEmFalhaCOM THEN
		stMotor.En.xSoftEmFalhaCOM := xSoftEmFalhaCOM;
	END_IF
		
	IF xFaltaDeFaseOk <> Ultima_stMotor.En.xFaltaDeFaseOk THEN
		stMotor.En.xFaltaDeFaseOk := xFaltaDeFaseOk;
	END_IF
	

END_IF




// quando mudam alguma coisa no st
IF stMotor.En.xEmergenciaOK <> Ultima_stMotor.En.xEmergenciaOK THEN
	xEmergenciaOK := stMotor.En.xEmergenciaOK;
END_IF

IF stMotor.En.xContatorLigado <> Ultima_stMotor.En.xContatorLigado THEN
	xContatorLigado := stMotor.En.xContatorLigado;
END_IF

IF stMotor.En.xDisjuntorOK <> Ultima_stMotor.En.xDisjuntorOK THEN
	xDisjuntorOK := stMotor.En.xDisjuntorOK;
END_IF

IF stMotor.En.xAutomaticoManual <> Ultima_stMotor.En.xAutomaticoManual THEN
	xAutomaticoManual := stMotor.En.xAutomaticoManual;
END_IF

IF stMotor.En.xBloqueado <> Ultima_stMotor.En.xBloqueado THEN
	xBloqueado := stMotor.En.xBloqueado;
END_IF

IF stMotor.En.iSenhaBloqueio <> Ultima_stMotor.En.iSenhaBloqueio THEN
	iSenhaBloqueio := stMotor.En.iSenhaBloqueio;
END_IF

IF stMotor.En.iSenhaAtual <> Ultima_stMotor.En.iSenhaAtual THEN
	iSenhaAtual := stMotor.En.iSenhaAtual;
END_IF

IF stMotor.En.xReversoAuto <> Ultima_stMotor.En.xReversoAuto THEN
	xReversoAuto := stMotor.En.xReversoAuto;
END_IF

IF stMotor.En.xLigaAuto <> Ultima_stMotor.En.xLigaAuto THEN
	xLigaAuto := stMotor.En.xLigaAuto;
END_IF

IF stMotor.En.xLigaManu <> Ultima_stMotor.En.xLigaManu THEN
	xLigaManu := stMotor.En.xLigaManu;
END_IF

IF stMotor.En.xReversoManu <> Ultima_stMotor.En.xReversoManu THEN
	xReversoManu := stMotor.En.xReversoManu;
END_IF

IF stMotor.En.xLigaManu3S <> Ultima_stMotor.En.xLigaManu3S THEN
	xLigaManu3S := stMotor.En.xLigaManu3S;
END_IF

IF stMotor.En.xReset <> Ultima_stMotor.En.xReset THEN
	xReset := stMotor.En.xReset;
END_IF

IF stMotor.En.xResetRegistros <> Ultima_stMotor.En.xResetRegistros THEN
	xResetRegistros := stMotor.En.xResetRegistros;
END_IF

IF stMotor.En.xInterLock_1 <> Ultima_stMotor.En.xInterLock_1 THEN
	xInterLock_1 := stMotor.En.xInterLock_1;
END_IF

IF stMotor.En.sInterLock_1 <> Ultima_stMotor.En.sInterLock_1 THEN
	sInterLock_1 := stMotor.En.sInterLock_1;
END_IF

IF stMotor.En.xInterLock_2 <> Ultima_stMotor.En.xInterLock_2 THEN
	xInterLock_2 := stMotor.En.xInterLock_2;
END_IF

IF stMotor.En.sInterLock_2 <> Ultima_stMotor.En.sInterLock_2 THEN
	sInterLock_2 := stMotor.En.sInterLock_2;
END_IF

IF stMotor.En.xInterLock_3 <> Ultima_stMotor.En.xInterLock_3 THEN
	xInterLock_3 := stMotor.En.xInterLock_3;
END_IF

IF stMotor.En.sInterLock_3 <> Ultima_stMotor.En.sInterLock_3 THEN
	sInterLock_3 := stMotor.En.sInterLock_3;
END_IF

IF stMotor.En.xInterLock_4 <> Ultima_stMotor.En.xInterLock_4 THEN
	xInterLock_4 := stMotor.En.xInterLock_4;
END_IF

IF stMotor.En.sInterLock_4 <> Ultima_stMotor.En.sInterLock_4 THEN
	sInterLock_4 := stMotor.En.sInterLock_4;
END_IF

IF stMotor.En.xTemInversor <> Ultima_stMotor.En.xTemInversor THEN
	xTemInversor := stMotor.En.xTemInversor;
END_IF

IF stMotor.En.xTemTeSysU <> Ultima_stMotor.En.xTemTeSysU THEN
	xTemTeSysU := stMotor.En.xTemTeSysU;
END_IF

IF stMotor.En.xInversorOnline <> Ultima_stMotor.En.xInversorOnline THEN
	xInversorOnline := stMotor.En.xInversorOnline;
END_IF

IF stMotor.En.xFalhaInversor <> Ultima_stMotor.En.xFalhaInversor THEN
	xFalhaInversor := stMotor.En.xFalhaInversor;
END_IF

IF stMotor.En.stHoraAgora.wMilliseconds <> Ultima_stMotor.En.stHoraAgora.wMilliseconds THEN
	stHoraAgora := stMotor.En.stHoraAgora;
END_IF

IF stMotor.En.xFazendoComissionamento <> Ultima_stMotor.En.xFazendoComissionamento THEN
	xFazendoComissionamento := stMotor.En.xFazendoComissionamento;
END_IF

IF stMotor.En.xFreioOK <> Ultima_stMotor.En.xFreioOK THEN
	xFreioOK := stMotor.En.xFreioOK;
END_IF

IF stMotor.En.xContatoInversorOK <> Ultima_stMotor.En.xContatoInversorOK THEN
	xContatoInversorOK := stMotor.En.xContatoInversorOK;
END_IF

IF stMotor.En.xContatoFalhaSoft <> Ultima_stMotor.En.xContatoFalhaSoft THEN
	xContatoFalhaSoft := stMotor.En.xContatoFalhaSoft;
END_IF

IF stMotor.En.xContatoRodandoSoft <> Ultima_stMotor.En.xContatoRodandoSoft THEN
	xContatoRodandoSoft := stMotor.En.xContatoRodandoSoft;
END_IF

IF stMotor.En.xSoftOnline <> Ultima_stMotor.En.xSoftOnline THEN
	xSoftOnline := stMotor.En.xSoftOnline;
END_IF

IF stMotor.En.xUsaVeloAuto2 <> Ultima_stMotor.En.xUsaVeloAuto2 THEN
	xUsaVeloAuto2 := stMotor.En.xUsaVeloAuto2;
END_IF

IF stMotor.En.xLigaHigienizacao <> Ultima_stMotor.En.xLigaHigienizacao THEN
	xLigaHigienizacao := stMotor.En.xLigaHigienizacao;
END_IF

IF stMotor.En.xResetaNumeroDeReset <> Ultima_stMotor.En.xResetaNumeroDeReset THEN
	xResetaNumeroDeReset := stMotor.En.xResetaNumeroDeReset;
END_IF

IF stMotor.En.xLocal <> Ultima_stMotor.En.xLocal THEN
	xLocal := stMotor.En.xLocal;
END_IF

IF stMotor.En.xContatoInversorOK <> Ultima_stMotor.En.xContatoInversorOK THEN
	xContatoInversorOK := stMotor.En.xContatoInversorOK;
END_IF

IF stMotor.En.xECO <> Ultima_stMotor.En.xECO THEN
	xECO := stMotor.En.xECO;
END_IF

IF stMotor.En.xResetBlocoComunicacao <> Ultima_stMotor.En.xResetBlocoComunicacao THEN
	xResetBlocoComunicacao := stMotor.En.xResetBlocoComunicacao;
END_IF

IF stMotor.En.xSoftEmFalhaCOM <> Ultima_stMotor.En.xSoftEmFalhaCOM THEN
	xSoftEmFalhaCOM := stMotor.En.xSoftEmFalhaCOM;
END_IF

IF stMotor.En.xFaltaDeFaseOk <> Ultima_stMotor.En.xFaltaDeFaseOk THEN
	xFaltaDeFaseOk := stMotor.En.xFaltaDeFaseOk;
END_IF




// salva oq tem pra proximo ciclo
//Ultima_stMotor := stMotor; essa linha consome muita CPU 

Ultima_stMotor.En := stMotor.En;
Ultima_stMotor.Config := stMotor.Config;
END_ACTION

ACTION AjustaSaida:

// oq é gerado aqui dentro tem que colocar pra jogar na saida
stMotor.Sa.xLigado				:= xLigado;
stMotor.Sa.xCmdFwd				:= xCmdFwd;
stMotor.Sa.xCmdRev				:= xCmdRev;
stMotor.Sa.xTrocandoSentido		:= xTrocandoSentido;
stMotor.Sa.xParadoPorInterlock	:= xParadoPorInterlock;
stMotor.Sa.iVelocidade			:= iVelocidade;
stMotor.Sa.iStsMotor			:= iStsMotor;
stMotor.Sa.xResetParaInversor	:= xResetParaInversor;
stMotor.Sa.xFalha				:= xFalha;
stMotor.Sa.iDisjDesarm			:= iDisjDesarm;
stMotor.Sa.iPartidas			:= iPartidas;
stMotor.Sa.iFalhaPartida		:= iFalhaPartida;
stMotor.Sa.xNaoLigaProxMotor	:= xNaoLigaProxMotor;
sNome_Funcao					:= stMotor.Config.sNome_Funcao;
stMotor.Sa.xFalhaContatora		:= xFalhaContatora;
stMotor.Sa.sStatus				:= sStatus;

// oq é gerado la fora tem que ser o inverso
rVoltagemEntrada	:= stMotor.Sa.rVoltagemEntrada;
rTorque				:= stMotor.Sa.rTorque;
rTemperaturaInver	:= stMotor.Sa.rTemperaturaInver;
rTemperaturaMotor	:= stMotor.Sa.rTemperaturaMotor;
rCorrente			:= stMotor.Sa.rCorrente;
rVelocidadeRPM		:= stMotor.Sa.rVelocidadeRPM;
rVelocidadeHz		:= stMotor.Sa.rVelocidadeHz;
sUltimoErro			:= stMotor.Sa.sUltimoErro;
sStatusConexao		:= stMotor.Sa.sStatusConexao;

//Estes so podem mudar na st pq ela é retentiva 

stMotor.Config.xTudoComissionado :=
	stMotor.Config.xComissionado_Corrente AND stMotor.Config.xComissionado_Sentido AND stMotor.Config.xComissionado_Velo;

xTudoComissionado := stMotor.Config.xTudoComissionado;

xComissionado_Sentido		:= stMotor.Config.xComissionado_Sentido;
xInverteSentido				:= stMotor.Config.xInverteSentido;
xVeloEmPorcentagem			:= stMotor.Config.xVeloEmPorcentagem;
rVeloEmPorcentagem_VeloMax	:= stMotor.Config.rVeloEmPorcentagem_VeloMax;
xVeloEmMetroPMin			:= stMotor.Config.xVeloEmMetroPMin;
rVeloEmMetroPMin_Conversao	:= stMotor.Config.rVeloEmMetroPMin_Conversao;
xComissionado_Velo			:= stMotor.Config.xComissionado_Velo;
xComissionado_Corrente		:= stMotor.Config.xComissionado_Corrente;
END_ACTION

ACTION AlarmesIHM:


FOR i := 0 TO 20 DO
	stMotor.ErrosIHM[i].xErro := FALSE;
	stMotor.ErrosIHM[i].Mensagem := '';
END_FOR



iaux := 0;
stMotor.ErrosIHM[iaux].xErro := NOT xEmergenciaOK;
stMotor.ErrosIHM[iaux].sTag := 'ucFalhaEmergência';
//coloca o nome da emergencia que esta precionada quando ele ta em emergencia, mas se nao tiver nome so escreve emergencia precionada
IF stMotor.ErrosIHM[iaux].xErro THEN
	FOR i := 1 TO 4 DO
		IF NOT stMotor.LeiturasInversorIHM.xStatusEmergencias[i] THEN
			CASE i OF
				1:stMotor.ErrosIHM[iaux].Mensagem := stMotor.BancoDeDados.Emerg1;
				2:stMotor.ErrosIHM[iaux].Mensagem := stMotor.BancoDeDados.Emerg2;
				3:stMotor.ErrosIHM[iaux].Mensagem := stMotor.BancoDeDados.Emerg3;
				4:stMotor.ErrosIHM[iaux].Mensagem := stMotor.BancoDeDados.Emerg4;
			END_CASE
			EXIT;
		END_IF
		IF stMotor.ErrosIHM[iaux].Mensagem = '' THEN
			stMotor.ErrosIHM[iaux].Mensagem := 'Emergência Pressionada';
		END_IF
	END_FOR
ELSE
	stMotor.ErrosIHM[iaux].Mensagem := 'Emergencia OK';
END_IF
iaux := iaux + 1;


stMotor.ErrosIHM[iaux].xErro := NOT xFaltaDeFaseOk;
stMotor.ErrosIHM[iaux].sTag := 'ucFaltaDeFase';
//coloca o nome da emergencia que esta precionada quando ele ta em emergencia, mas se nao tiver nome so escreve emergencia precionada
IF stMotor.ErrosIHM[iaux].xErro THEN
	IF stMotor.ErrosIHM[iaux].Mensagem = '' THEN
		stMotor.ErrosIHM[iaux].Mensagem := 'Falta de fase';
	END_IF
ELSE
	stMotor.ErrosIHM[iaux].Mensagem := 'Fase OK';
END_IF
iaux := iaux + 1;

IF xTemContatora THEN
	stMotor.ErrosIHM[iaux].xErro := xFalhaContatora;
	stMotor.ErrosIHM[iaux].sTag := 'ucFalhaContatora';
	IF stMotor.ErrosIHM[iaux].xErro THEN
		stMotor.ErrosIHM[iaux].Mensagem := 'Erro Contatora';
	ELSE
		stMotor.ErrosIHM[iaux].Mensagem := 'Contatora OK';
	END_IF
	iaux := iaux + 1;
END_IF

IF xTemDisjuntor THEN
	stMotor.ErrosIHM[iaux].xErro := NOT xDisjuntorOK AND NOT xByPassDisjuntor;
	stMotor.ErrosIHM[iaux].sTag := 'ucFalhaDisjuntor';
	IF stMotor.ErrosIHM[iaux].xErro THEN
		stMotor.ErrosIHM[iaux].Mensagem := 'Disjuntor Desarmado';
	ELSE
		stMotor.ErrosIHM[iaux].Mensagem := 'Disjuntor OK';
	END_IF
	iaux := iaux + 1;
END_IF

IF xTemInversor THEN
	stMotor.ErrosIHM[iaux].xErro := (xTemInversor AND (NOT xInversorOnline AND NOT xBypassRede));
	stMotor.ErrosIHM[iaux].sTag := 'ucFalhaInversorOffline';
	IF stMotor.ErrosIHM[iaux].xErro THEN
		stMotor.ErrosIHM[iaux].Mensagem := 'Inversor Offline';
	ELSE
		stMotor.ErrosIHM[iaux].Mensagem := 'Inversor Online';
	END_IF
	iaux := iaux + 1;
END_IF

IF xTemInversor THEN
	stMotor.ErrosIHM[iaux].xErro := (xTemInversor AND (xFalhaInversor AND NOT xBypassRede));
	stMotor.ErrosIHM[iaux].sTag := 'ucFalhaInversor';
	IF stMotor.ErrosIHM[iaux].xErro THEN
		stMotor.ErrosIHM[iaux].Mensagem := 'Inversor falha';
	ELSE
		stMotor.ErrosIHM[iaux].Mensagem := 'Inversor OK';
	END_IF
	iaux := iaux + 1;
END_IF

IF xTemTeSysU THEN
	stMotor.ErrosIHM[iaux].xErro := (xTemTeSysU AND (NOT xInversorOnline AND NOT xBypassRede));
	stMotor.ErrosIHM[iaux].sTag := 'ucFalhaInversorOffline';
	IF stMotor.ErrosIHM[iaux].xErro THEN
		stMotor.ErrosIHM[iaux].Mensagem := 'TeSysU Offline';
	ELSE
		stMotor.ErrosIHM[iaux].Mensagem := 'TeSysU Online';
	END_IF
	iaux := iaux + 1;
END_IF

IF xTemTeSysU THEN
	stMotor.ErrosIHM[iaux].xErro := (xTemTeSysU AND (xFalhaInversor AND NOT xBypassRede));
	stMotor.ErrosIHM[iaux].sTag := 'ucFalhaInversor';
	IF stMotor.ErrosIHM[iaux].xErro THEN
		stMotor.ErrosIHM[iaux].Mensagem := 'TeSysU falha';
	ELSE
		stMotor.ErrosIHM[iaux].Mensagem := 'TeSysU OK';
	END_IF
	iaux := iaux + 1;
END_IF

IF xTemContatoInversorOK THEN
	stMotor.ErrosIHM[iaux].xErro := (xTemContatoInversorOK AND (NOT (xContatoInversorOK) AND NOT xBypassContatoInversorOK));
	stMotor.ErrosIHM[iaux].sTag := 'ucFalhaContatoInversor';
	IF stMotor.ErrosIHM[iaux].xErro THEN
		stMotor.ErrosIHM[iaux].Mensagem := 'Contato inversor falha';
	ELSE
		stMotor.ErrosIHM[iaux].Mensagem := 'Contato inversor OK';
	END_IF
	iaux := iaux + 1;
END_IF

IF stMotor.Config.xTemFreio THEN
	stMotor.ErrosIHM[iaux].xErro := (stMotor.Config.xTemFreio AND (NOT xFreioOK AND NOT xBypassFreio));
	stMotor.ErrosIHM[iaux].sTag := 'ucFalhaFreio';
	IF stMotor.ErrosIHM[iaux].xErro THEN
		stMotor.ErrosIHM[iaux].Mensagem := 'Freio Desarmado';
	ELSE
		stMotor.ErrosIHM[iaux].Mensagem := 'Freio OK';
	END_IF
	iaux := iaux + 1;
END_IF

IF stMotor.Config.xTemSoft THEN
	stMotor.ErrosIHM[iaux].xErro := ((xContatoFalhaSoft AND NOT  xBypassContatoFalhaSoft) OR (xSoftEmFalhaCOM AND NOT xBypassSoftEmFalhaCOM)) AND stMotor.Config.xTemSoft;
	stMotor.ErrosIHM[iaux].sTag := 'ucFalhaSoft';
	IF stMotor.ErrosIHM[iaux].xErro THEN
		stMotor.ErrosIHM[iaux].Mensagem := 'Soft em falha';
	ELSE
		stMotor.ErrosIHM[iaux].Mensagem := 'Soft OK';
	END_IF
	iaux := iaux + 1;
END_IF

IF stMotor.Config.xTemSoft THEN
	stMotor.ErrosIHM[iaux].xErro := ((xFalhaPartidaSoft AND NOT xBypassContatoRunSoft)) AND stMotor.Config.xTemSoft;
	stMotor.ErrosIHM[iaux].sTag := 'ucFalhaSoft';
	IF stMotor.ErrosIHM[iaux].xErro THEN
		stMotor.ErrosIHM[iaux].Mensagem := 'Falha partida Soft';
	ELSE
		IF NOT (xCmdFwd OR xCmdRev) THEN
			stMotor.ErrosIHM[iaux].Mensagem := 'Parada';
		ELSIF NOT xFalhaPartidaSoft AND NOT xContatoRodandoSoft THEN
			stMotor.ErrosIHM[iaux].Mensagem := 'Partindo';
		ELSE
			stMotor.ErrosIHM[iaux].Mensagem := 'Partiu';
		END_IF
	END_IF
	iaux := iaux + 1;
END_IF
END_ACTION

ACTION Contagem:

// contagens
rtSucessonaPartida(CLK := ((iStsMotor = 3 OR iStsMotor = 4) AND (((xContatorLigado OR xByPassContator)) AND xTemContatora OR NOT xTemContatora)), Q =>);
IF rtSucessonaPartida.q THEN
	iPartidas := iPartidas + 1;
END_IF


rtDisjuntorDesarmado(CLK := iStsMotor = 8, Q =>);
IF rtDisjuntorDesarmado.q THEN
	iDisjDesarm := iDisjDesarm + 1;
END_IF


rtFalhanaPartida(CLK := xFalha, Q =>);
IF rtFalhanaPartida.q THEN
	iFalhaPartida := iFalhaPartida + 1;
END_IF


IF xResetRegistros THEN
	iFalhaPartida	:= 0;
	iDisjDesarm		:= 0;
	iPartidas		:= 0;
END_IF
END_ACTION

ACTION ControleBloqueio:

rtDesbloquiou(CLK := xBloqueado, Q =>);

IF rtDesbloquiou.q THEN
	IF (iSenhaBloqueio <> iSenhaAtual) THEN
		xBloqueado := TRUE;
	ELSE
		iSenhaBloqueio	:= 0;
		iSenhaAtual		:= 0;
	END_IF
END_IF

rtBloqueiou(CLK := xBloqueado, Q =>);

IF rtBloqueiou.q THEN
	iSenhaBloqueio	:= iSenhaAtual;
	iSenhaAtual		:= 0;
END_IF
END_ACTION

ACTION ControleDaPartida:

// INICIO CONTROLE AUTOMATICO MANUAL

//Bloqueio caso de emergencia e ele esteja em manual, ai ele nao religa sozinho quando sair a emergencia mas no em manual
rtTavaEmEmergencia(CLK := NOT xEmergenciaOK AND NOT xAutomaticoManual AND xLigaManu, Q =>);

IF rtTavaEmEmergencia.q THEN
	xTavaEmEmergencia := TRUE;
END_IF

rtVoltaEmergencia(CLK := xEmergenciaOK AND NOT xLigaManu, Q =>);

IF rtVoltaEmergencia.q THEN
	xTavaEmEmergencia := FALSE;
END_IF

//quando trocar de automatico pra manual ele desliga o manual
ftManual(CLK := xAutomaticoManual, Q =>);

IF ftManual.q THEN
	xLigaManu := FALSE;
END_IF

//Controle do liga 3 segundos

Ton3Segundos(IN := xLigaManu3S, PT := T#3S, Q =>, ET =>);
IF Ton3Segundos.q THEN
	//xLigaManu3S := FALSE;
END_IF

//controle da partida
xParadoPorInterlock := FALSE;

//Ve as emergencias dele
IF xEmergenciaOK THEN
	//se nao tiver bloqueado
	IF NOT xBloqueado THEN
		//tudo que da pra considerar uma falha
		IF (NOT xFalha) THEN
			//o controle se tudo tiver certo
			IF xAutomaticoManual THEN //Automatico
				IF NOT xLigaHigienizacao THEN
					IF xLigaAuto THEN
						// olha os interlocks e a reversao e o ECO
						IF NOT (xInterLock_1 OR xInterLock_2 OR xInterLock_3 OR xInterLock_4 OR xECO) THEN
							IF stMotor.Config.xTemReversao THEN
								xCmdFWD	:= NOT xReversoAuto;
								xCmdRev	:= xReversoAuto;
							ELSE
								xCmdFWD := TRUE;
							END_IF
	
							xParadoPorInterlock := FALSE;
						ELSE
							xCmdFWD := xCmdRev	:= FALSE;
							xParadoPorInterlock	:= TRUE;
						END_IF
					ELSE
						xCmdFWD := xCmdRev := FALSE;
					END_IF
				ELSE// se tiver com higienização ele liga a esteira
					xCmdFWD := xHabilitaHigienizacao;
				END_IF	
			ELSE // manual
				IF (xLigaManu OR (xLigaManu3S AND NOT Ton3Segundos.q)) AND NOT xTavaEmEmergencia THEN
					IF stMotor.Config.xTemReversao THEN
						xCmdFWD	:= NOT xReversoManu;
						xCmdRev	:= xReversoManu;
					ELSE
						xCmdFWD := TRUE;
					END_IF
				ELSE
					xCmdFWD := xCmdRev := FALSE;
				END_IF
			END_IF
		ELSE
			xCmdFWD := xCmdRev := FALSE;
		END_IF
	ELSE
		xCmdFWD := FALSE;
	END_IF
ELSE
	xCmdFWD := xCmdRev := FALSE;
END_IF

IF (xReset OR xResetBlocoComunicacao) AND xFalha THEN
	xCmdFWD := xCmdRev := FALSE;
END_IF

xLigado := xCmdFwd OR xCmdRev OR xParadoPorInterlock;
END_ACTION

ACTION ControleReset:





rtReset(CLK:= xReset AND xFalha, Q=> );
IF rtReset.Q THEN
	stMotor.En.iNumeroDeReset := stMotor.En.iNumeroDeReset + 1;
END_IF


IF (stMotor.En.iNumeroDeReset > stMotor.Config.iLimiteReset) AND stMotor.Config.xTemLimiteReset THEN
	xReset := FALSE;
END_IF


IF stMotor.En.xResetaNumeroDeReset THEN
	stMotor.En.xResetaNumeroDeReset := FALSE;
	stMotor.En.iNumeroDeReset := 0;
END_IF


tonResetFalha(IN := stMotor.En.iNumeroDeReset > 0 AND NOT xFalha, PT := ULINT_TO_TIME(stMotor.Config.iMinBloqueio*1000*60), Q =>, ET =>);
IF tonResetFalha.q THEN
	stMotor.En.xResetaNumeroDeReset := TRUE;
END_IF
END_ACTION

ACTION ControleVelocidade:

//Controle da velocidade

//se tiver comissionado ele ajeita a velo automatica pra ficar certo na saida
IF stMotor.Config.xComissionado_Velo THEN
	
	IF xUsaVeloAuto2 THEN
		iVelocidade := REAL_TO_INT(rSetPoinAuto2);
	ELSE
		iVelocidade := REAL_TO_INT(rSetPoinAuto);
	END_IF

	//protege contra numeros negativos ou divisao por 0
	IF stMotor.Config.xVeloEmPorcentagem THEN
		IF stMotor.Config.rVeloEmPorcentagem_VeloMax < 0.1 THEN
			stMotor.Config.rVeloEmPorcentagem_VeloMax := 1;
		END_IF
		IF xAutomaticoManual THEN
			IF xLigaHigienizacao THEN
				iVelocidade := REAL_TO_INT(rPorcentagemHigienizacao*(rSetPoinAuto * rPorcentagemHigienizacao * stMotor.Config.rVeloEmPorcentagem_VeloMax) / 100);
			ELSE
				IF xUsaVeloAuto2 THEN
					iVelocidade := REAL_TO_INT((rSetPoinAuto2 * stMotor.Config.rVeloEmPorcentagem_VeloMax) / 100);
				ELSE
					iVelocidade := REAL_TO_INT((rSetPoinAuto * stMotor.Config.rVeloEmPorcentagem_VeloMax) / 100);
				END_IF
			END_IF
		ELSE
			iVelocidade := REAL_TO_INT((rSetPoinManu * stMotor.Config.rVeloEmPorcentagem_VeloMax) / 100);
		END_IF
		
	END_IF

	IF stMotor.Config.xVeloEmMetroPMin THEN
		//protege contra numeros negativos ou divisao por 0
		IF stMotor.Config.rVeloEmMetroPMin_Conversao < 0.1 THEN
			stMotor.Config.rVeloEmMetroPMin_Conversao := 1;
		END_IF
		IF xAutomaticoManual THEN
			IF xLigaHigienizacao THEN
					iVelocidade := REAL_TO_INT(rPorcentagemHigienizacao*(rSetPoinAuto * 1800 / stMotor.Config.rVeloEmMetroPMin_Conversao));
			ELSE
				IF xUsaVeloAuto2 THEN
					iVelocidade := REAL_TO_INT((rSetPoinAuto2 * 1800 / stMotor.Config.rVeloEmMetroPMin_Conversao));
				ELSE
					iVelocidade := REAL_TO_INT((rSetPoinAuto * 1800 / stMotor.Config.rVeloEmMetroPMin_Conversao));				
				END_IF
			END_IF
		ELSE
			rAux := rSetPoinManu * 1800 / stMotor.Config.rVeloEmMetroPMin_Conversao;
			iVelocidade := REAL_TO_INT(rAux);
		END_IF
		
		
	END_IF
ELSE
	IF xAutomaticoManual THEN
		//se for higienização ele roda em 10%
		IF xLigaHigienizacao THEN
			iVelocidade := REAL_TO_INT(rPorcentagemHigienizacao*(rSetPoinAuto));
		ELSE
			//controla as 2 velo 
			IF xUsaVeloAuto2 THEN
				iVelocidade := REAL_TO_INT((rSetPoinAuto2));
			ELSE
				iVelocidade := REAL_TO_INT((rSetPoinAuto));
			END_IF
		END_IF
	ELSE
		iVelocidade := REAL_TO_INT(rSetPoinManu);
	END_IF
END_IF


//Se a regra de 3 der overflow aqui ele garante que nao vai girar pro lado errado
IF iVelocidade < 0 THEN
	iVelocidade := 0;
END_IF


//independende do automatico ou do munual ele roda sempre pro msm lado
// se tiver que inverte a velo e tiver comissionado
IF stMotor.Config.xInverteSentido AND (stMotor.Config.xComissionado_Sentido) THEN
	//se o operador meter uma velo negativa nao da BO
	IF iVelocidade < 0 THEN
		iVelocidade := iVelocidade;
	ELSE
		iVelocidade := iVelocidade * -1;
	END_IF
END_IF
END_ACTION

ACTION EmComissionamento:

xAutomaticoManual	:= FALSE;
//rSetPoinManu		:= 1800;
xReversoManu		:= FALSE;

Ton3Segundos(IN := xLigaManu3S, PT := T#3S, Q =>, ET =>);

IF Ton3Segundos.q THEN
	xLigaManu3S := FALSE;
END_IF

